  MoveC 1160 to (433.16, -30.09, -5) mm, rotated rx -180 ry 0 rz 30 deg; joints [33.705, -53.903, 150.227, 63.755, -91.912, 5.472] to (420.46, -17.39, -5) mm, rotated rx -180 ry 0 rz 30 deg; joints [33.923, -53.753, 148.985, 63.944, -91.411, 4.501]
  MoveL 1161 to (395.06, -17.39, -5) mm, rotated rx -180 ry 0 rz 0 deg; joints [25.034, -53.985, 155.724, 25.42, -99.757, 5.283]
  MoveL 1162 to (318.86, -17.39, -5) mm, rotated rx -180 ry 0 rz 0 deg; joints [22.969, -53.773, 150.895, 23.082, -95.687, 3.059]
  MoveC 1163 to (306.16, -30.09, -5) mm, rotated rx -180 ry 0 rz 0 deg; joints [21.911, -53.706, 150.409, 22.005, -95.348, 2.779] to (293.46, -17.39, -5) mm, rotated rx -180 ry 0 rz 0 deg; joints [22.351, -53.577, 149.245, 22.413, -94.372, 2.431]
  MoveL 1164 to (191.86, -17.39, -5) mm, rotated rx -180 ry 0 rz 0 deg; joints [20.165, -52.294, 142.446, 20.16, -89.274, 0.325]
  MoveC 1165 to (179.16, -30.09, -5) mm, rotated rx -180 ry 0 rz 0 deg; joints [19.25, -52.149, 141.884, 19.247, -88.88, 0.185] to (166.46, -17.39, -5) mm, rotated rx -180 ry 0 rz 0 deg; joints [19.681, -51.866, 140.698, 19.687, -88.03, -0.121]
  MoveL 1166 to (90.26, -17.39, -5) mm, rotated rx -180 ry 0 rz 0 deg; joints [18.355, -50.37, 135.332, 18.442, -84.349, -1.32]
  MoveL 1167 to (64.86, -17.39, -5) mm, rotated rx 180 ry 0 rz 0 deg; joints [17.951, -49.807, 133.502, 18.078, -83.134, -1.681]
  MoveC 1168 to (61.14, -26.37, -5) mm, rotated rx 180 ry 0 rz 0 deg; joints [17.461, -49.78, 133.439, 17.587, -83.082, -1.64] to (52.16, -30.09, -5) mm, rotated rx -180 ry 0 rz 0 deg; joints [17.147, -49.597, 132.868, 17.286, -82.702, -1.723]
  MoveL 1169 to (52.16, -30.09, -5) mm, rotated rx -180 ry 0 rz 0 deg; joints [17.147, -49.597, 132.868, 17.286, -82.702, -1.723]
  MoveC 1170 to (43.18, -26.37, -5) mm, rotated rx -180 ry 0 rz 0 deg; joints [17.193, -49.362, 132.128, 17.351, -82.221, -1.88] to (39.46, -17.39, -5) mm, rotated rx -180 ry 0 rz 0 deg; joints [17.563, -49.213, 131.65, 17.739, -81.923, -2.026]
  MoveL 1171 to (14.06, -17.39, -5) mm, rotated rx 180 ry 0 rz 0 deg; joints [17.191, -48.59, 129.776, 17.421, -80.714, -2.357]
  MoveC 1172 to (13.61, -17.2, -5) mm, rotated rx -180 ry 0 rz 0 deg; joints [17.194, -48.578, 129.738, 17.424, -80.69, -2.365] to (13.42, -16.75, -5) mm, rotated rx 180 ry 0 rz 0 deg; joints [17.212, -48.57, 129.714, 17.443, -80.675, -2.373]
  MoveL 1173 to (13.42, -16.12, -5) mm, rotated rx 180 ry 0 rz 0 deg; joints [17.241, -48.565, 129.7, 17.474, -80.667, -2.38]
  MoveC 1174 to (13.42, -15.67, -4.81) mm, rotated rx -180 ry 0 rz 0 deg; joints [17.262, -48.576, 129.692, 17.495, -80.65, -2.389] to (13.42, -15.48, -4.37) mm, rotated rx 180 ry 0 rz 0 deg; joints [17.27, -48.607, 129.693, 17.505, -80.622, -2.399]
  Set speed (1000.0 mm/s)
  MoveL 1175 to (13.42, -15.48, 5) mm, rotated rx -180 ry 0 rz 0 deg; joints [17.266, -49.29, 129.811, 17.53, -80.082, -2.572]
  MoveL 1176 to (12.15, -16.75, 5) mm, rotated rx -180 ry 0 rz 0 deg; joints [17.189, -49.267, 129.745, 17.454, -80.039, -2.572]
  Set speed (25.4 mm/s)
  MoveL 1177 to (12.15, -16.75, 1) mm, rotated rx -180 ry 0 rz 0 deg; joints [17.191, -48.975, 129.696, 17.443, -80.27, -2.499]
  MoveL 1178 to (12.15, -16.75, -7.72) mm, rotated rx -180 ry 0 rz 0 deg; joints [17.195, -48.34, 129.584, 17.421, -80.77, -2.34]
  MoveC 1179 to (12.34, -16.75, -8.16) mm, rotated rx -180 ry 0 rz 0 deg; joints [17.198, -48.312, 129.592, 17.422, -80.804, -2.33] to (12.79, -16.75, -8.35) mm, rotated rx -180 ry 0 rz 0 deg; joints [17.204, -48.309, 129.623, 17.427, -80.836, -2.32]
  Set speed (50.8 mm/s)
  MoveL 1180 to (13.42, -16.75, -8.35) mm, rotated rx 180 ry 0 rz 0 deg; joints [17.213, -48.325, 129.67, 17.435, -80.867, -2.312]
  MoveC 1181 to (13.87, -16.94, -8.35) mm, rotated rx 180 ry 0 rz 0 deg; joints [17.211, -48.337, 129.708, 17.432, -80.891, -2.304] to (14.06, -17.39, -8.35) mm, rotated rx -180 ry 0 rz 0 deg; joints [17.193, -48.345, 129.732, 17.412, -80.905, -2.297]
  MoveL 1182 to (14.06, -169.79, -8.35) mm, rotated rx 180 ry 0 rz 0 deg; joints [9.89, -49.145, 132.47, 9.97, -82.555, -0.881]
  MoveL 1183 to (471.26, -169.79, -8.35) mm, rotated rx 180 ry 0 rz 30 deg; joints [26.891, -53.506, 157.289, 57.471, -96.607, 11.391]
  MoveL 1184 to (471.26, -17.39, -8.35) mm, rotated rx 180 ry 0 rz 30 deg; joints [35.771, -53.739, 151.859, 65.871, -92.441, 7.208]
  MoveL 1185 to (445.86, -17.39, -8.35) mm, rotated rx 180 ry 0 rz 30 deg; joints [34.827, -53.598, 150.406, 64.887, -92.006, 5.964]
  MoveC 1186 to (433.16, -30.09, -8.35) mm, rotated rx -180 ry 0 rz 30 deg; joints [33.707, -53.551, 150.167, 63.767, -92.041, 5.734] to (420.46, -17.39, -8.35) mm, rotated rx -180 ry 0 rz 30 deg; joints [33.926, -53.411, 148.927, 63.953, -91.536, 4.756]
  MoveL 1187 to (395.06, -17.39, -8.35) mm, rotated rx -180 ry 0 rz 0 deg; joints [25.037, -53.585, 155.656, 25.448, -100.057, 5.428]
  MoveL 1188 to (318.86, -17.39, -8.35) mm, rotated rx -180 ry 0 rz 0 deg; joints [22.971, -53.416, 150.834, 23.097, -95.959, 3.176]
  MoveC 1189 to (306.16, -30.09, -8.35) mm, rotated rx 180 ry 0 rz 0 deg; joints [21.913, -53.353, 150.349, 22.018, -95.619, 2.89] to (293.46, -17.39, -8.35) mm, rotated rx -180 ry 0 rz 0 deg; joints [22.353, -53.232, 149.186, 22.423, -94.636, 2.54]
  MoveL 1190 to (191.86, -17.39, -8.35) mm, rotated rx 180 ry 0 rz 0 deg; joints [20.167, -51.993, 142.395, 20.161, -89.507, 0.411]
  MoveC 1191 to (179.16, -30.09, -8.35) mm, rotated rx -180 ry 0 rz 0 deg; joints [19.251, -51.851, 141.833, 19.247, -89.113, 0.266] to (166.46, -17.39, -8.35) mm, rotated rx -180 ry 0 rz 0 deg; joints [19.683, -51.575, 140.647, 19.686, -88.257, -0.04]
  MoveL 1192 to (90.26, -17.39, -8.35) mm, rotated rx -180 ry 0 rz 0 deg; joints [18.357, -50.104, 135.285, 18.436, -84.557, -1.25]
  MoveL 1193 to (64.86, -17.39, -8.35) mm, rotated rx -180 ry 0 rz 0 deg; joints [17.952, -49.548, 133.456, 18.072, -83.337, -1.614]
  MoveC 1194 to (61.14, -26.37, -8.35) mm, rotated rx -180 ry 0 rz 0 deg; joints [17.462, -49.522, 133.393, 17.581, -83.285, -1.576] to (52.16, -30.09, -8.35) mm, rotated rx -180 ry 0 rz 0 deg; joints [17.149, -49.341, 132.823, 17.279, -82.904, -1.66]
  MoveL 1195 to (52.16, -30.09, -8.35) mm, rotated rx -180 ry 0 rz 0 deg; joints [17.149, -49.341, 132.823, 17.279, -82.904, -1.66]
  MoveC 1196 to (43.18, -26.37, -8.35) mm, rotated rx -180 ry 0 rz 0 deg; joints [17.194, -49.108, 132.082, 17.344, -82.42, -1.818] to (39.46, -17.39, -8.35) mm, rotated rx -180 ry 0 rz 0 deg; joints [17.565, -48.961, 131.605, 17.731, -82.12, -1.963]
  MoveL 1197 to (14.06, -17.39, -8.35) mm, rotated rx 180 ry 0 rz 0 deg; joints [17.193, -48.345, 129.732, 17.412, -80.905, -2.297]
  MoveC 1198 to (13.61, -17.2, -8.35) mm, rotated rx -180 ry 0 rz 0 deg; joints [17.195, -48.333, 129.694, 17.416, -80.881, -2.305] to (13.42, -16.75, -8.35) mm, rotated rx 180 ry 0 rz 0 deg; joints [17.213, -48.325, 129.67, 17.435, -80.867, -2.312]
  MoveL 1199 to (13.42, -16.12, -8.35) mm, rotated rx -180 ry 0 rz 0 deg; joints [17.243, -48.32, 129.656, 17.465, -80.858, -2.32]
  MoveC 1200 to (13.42, -15.67, -8.16) mm, rotated rx -180 ry 0 rz 0 deg; joints [17.263, -48.331, 129.648, 17.487, -80.842, -2.328] to (13.42, -15.48, -7.72) mm, rotated rx -180 ry 0 rz 0 deg; joints [17.272, -48.362, 129.649, 17.497, -80.814, -2.338]
  Set speed (1000.0 mm/s)
  MoveL 1201 to (13.42, -15.48, 6) mm, rotated rx 180 ry 0 rz 0 deg; joints [17.266, -49.363, 129.823, 17.533, -80.024, -2.59]
  MoveL 1202 to (-18.41, -15.48, 6) mm, rotated rx -180 ry 0 rz 0 deg; joints [16.82, -48.516, 127.438, 17.166, -78.533, -2.979]
  Set speed (25.4 mm/s)
  MoveL 1203 to (-18.41, -15.48, -4.37) mm, rotated rx -180 ry 0 rz 0 deg; joints [16.824, -47.785, 127.311, 17.136, -79.111, -2.798]
  MoveC 1204 to (-18.41, -15.67, -4.81) mm, rotated rx -180 ry 0 rz 0 deg; joints [16.816, -47.754, 127.31, 17.126, -79.138, -2.788] to (-18.41, -16.12, -5) mm, rotated rx -180 ry 0 rz 0 deg; joints [16.795, -47.745, 127.318, 17.104, -79.154, -2.779]
  Set speed (50.8 mm/s)
  MoveL 1205 to (-18.41, -16.75, -5) mm, rotated rx -180 ry 0 rz 0 deg; joints [16.767, -47.749, 127.332, 17.074, -79.162, -2.771]
  MoveC 1206 to (-18.6, -17.2, -5) mm, rotated rx 180 ry 0 rz 0 deg; joints [16.744, -47.748, 127.328, 17.051, -79.158, -2.768] to (-19.04, -17.39, -5) mm, rotated rx -180 ry 0 rz 0 deg; joints [16.729, -47.737, 127.299, 17.037, -79.139, -2.771]
  MoveL 1207 to (-39.46, -17.39, -5) mm, rotated rx -180 ry 0 rz 0 deg; joints [16.456, -47.188, 125.751, 16.818, -78.168, -3.017]
  MoveC 1208 to (-52.16, -30.09, -5) mm, rotated rx 180 ry 0 rz 0 deg; joints [15.728, -46.931, 125.057, 16.101, -77.708, -2.999] to (-64.86, -17.39, -5) mm, rotated rx -180 ry 0 rz 0 deg; joints [16.128, -46.481, 123.801, 16.561, -76.959, -3.315]
  MoveL 1209 to (-90.26, -17.39, -5) mm, rotated rx -180 ry 0 rz 0 deg; joints [15.813, -45.748, 121.826, 16.323, -75.747, -3.606]
  MoveL 1210 to (-166.46, -17.39, -5) mm, rotated rx -180 ry 0 rz 0 deg; joints [14.935, -43.396, 115.729, 15.709, -72.082, -4.442]
  MoveC 1211 to (-179.16, -30.09, -5) mm, rotated rx 180 ry 0 rz 0 deg; joints [14.282, -43.083, 114.956, 15.064, -71.585, -4.366] to (-191.86, -17.39, -5) mm, rotated rx -180 ry 0 rz 0 deg; joints [14.663, -42.561, 113.635, 15.537, -70.846, -4.712]
  MoveL 1212 to (-293.46, -17.39, -5) mm, rotated rx -180 ry 0 rz 0 deg; joints [13.666, -38.954, 104.895, 15.006, -65.798, -5.788]
  MoveC 1213 to (-306.16, -30.09, -5) mm, rotated rx -180 ry 0 rz 0 deg; joints [13.075, -38.58, 104.026, 14.418, -65.257, -5.668] to (-318.86, -17.39, -5) mm, rotated rx -180 ry 0 rz 0 deg; joints [13.438, -37.982, 102.606, 14.913, -64.502, -6.06]
  MoveL 1214 to (-395.06, -17.39, -5) mm, rotated rx -180 ry 0 rz 0 deg; joints [12.794, -34.878, 95.441, 14.734, -60.499, -6.909]
  MoveL 1215 to (-420.46, -17.39, -5) mm, rotated rx -180 ry 0 rz 0 deg; joints [12.593, -33.776, 92.938, 14.71, -59.119, -7.208]
  MoveC 1216 to (-433.16, -30.09, -5) mm, rotated rx -180 ry 0 rz 0 deg; joints [12.054, -33.329, 91.94, 14.168, -58.516, -7.053] to (-445.86, -17.39, -5) mm, rotated rx 180 ry 0 rz 0 deg; joints [12.398, -32.635, 90.369, 14.706, -57.712, -7.518]
  MoveL 1217 to (-471.26, -17.39, -5) mm, rotated rx -180 ry 0 rz 0 deg; joints [12.209, -31.453, 87.727, 14.724, -56.273, -7.841]
  MoveL 1218 to (-471.26, -169.79, -5) mm, rotated rx 180 ry 0 rz 0 deg; joints [6.952, -32.605, 90.415, 8.272, -57.207, -4.124]
  MoveL 1219 to (-14.06, -169.79, -5) mm, rotated rx -180 ry 0 rz 0 deg; joints [9.653, -48.705, 130.382, 9.771, -80.926, -1.136]
  MoveL 1220 to (-14.06, -17.39, -5) mm, rotated rx 180 ry 0 rz 0 deg; joints [16.797, -47.869, 127.675, 17.093, -79.377, -2.71]
  MoveL 1221 to (-19.04, -17.39, -5) mm, rotated rx -180 ry 0 rz 0 deg; joints [16.729, -47.737, 127.299, 17.037, -79.139, -2.771]
  MoveC 1222 to (-19.49, -17.2, -5) mm, rotated rx -180 ry 0 rz 0 deg; joints [16.732, -47.724, 127.26, 17.041, -79.116, -2.779] to (-19.68, -16.75, -5) mm, rotated rx -180 ry 0 rz 0 deg; joints [16.749, -47.716, 127.236, 17.06, -79.101, -2.787]
  MoveL 1223 to (-19.68, -16.12, -5) mm, rotated rx -180 ry 0 rz 0 deg; joints [16.778, -47.711, 127.222, 17.09, -79.094, -2.795]
  MoveC 1224 to (-19.68, -15.67, -4.81) mm, rotated rx -180 ry 0 rz 0 deg; joints [16.798, -47.721, 127.214, 17.111, -79.078, -2.804] to (-19.68, -15.48, -4.37) mm, rotated rx -180 ry 0 rz 0 deg; joints [16.807, -47.751, 127.216, 17.121, -79.051, -2.814]
  Set speed (1000.0 mm/s)
  MoveL 1225 to (-19.68, -15.48, 5) mm, rotated rx -180 ry 0 rz 0 deg; joints [16.803, -48.411, 127.33, 17.149, -78.529, -2.977]
  MoveL 1226 to (-18.41, -15.48, 5) mm, rotated rx -180 ry 0 rz 0 deg; joints [16.82, -48.446, 127.426, 17.163, -78.589, -2.962]
  Set speed (25.4 mm/s)
  MoveL 1227 to (-18.41, -15.48, 1) mm, rotated rx -180 ry 0 rz 0 deg; joints [16.822, -48.164, 127.378, 17.151, -78.813, -2.892]
  MoveL 1228 to (-18.41, -15.48, -7.71) mm, rotated rx -180 ry 0 rz 0 deg; joints [16.825, -47.548, 127.268, 17.126, -79.296, -2.74]
  MoveC 1229 to (-18.41, -15.67, -8.16) mm, rotated rx -180 ry 0 rz 0 deg; joints [16.817, -47.518, 127.267, 17.116, -79.324, -2.73] to (-18.41, -16.12, -8.35) mm, rotated rx 180 ry 0 rz 0 deg; joints [16.797, -47.508, 127.275, 17.095, -79.339, -2.721]
  Set speed (50.8 mm/s)
  MoveL 1230 to (-18.41, -16.75, -8.35) mm, rotated rx -180 ry 0 rz 0 deg; joints [16.768, -47.512, 127.289, 17.065, -79.347, -2.714]
  MoveC 1231 to (-18.6, -17.2, -8.35) mm, rotated rx -180 ry 0 rz 0 deg; joints [16.745, -47.511, 127.285, 17.042, -79.344, -2.71] to (-19.04, -17.39, -8.35) mm, rotated rx -180 ry 0 rz 0 deg; joints [16.731, -47.5, 127.255, 17.028, -79.325, -2.713]
  MoveL 1232 to (-39.46, -17.39, -8.35) mm, rotated rx -180 ry 0 rz 0 deg; joints [16.458, -46.956, 125.708, 16.808, -78.35, -2.961]
  MoveC 1233 to (-52.16, -30.09, -8.35) mm, rotated rx 180 ry 0 rz 0 deg; joints [15.729, -46.701, 125.015, 16.091, -77.889, -2.946] to (-64.86, -17.39, -8.35) mm, rotated rx 180 ry 0 rz 0 deg; joints [16.13, -46.255, 123.76, 16.551, -77.136, -3.262]
  MoveL 1234 to (-90.26, -17.39, -8.35) mm, rotated rx -180 ry 0 rz 0 deg; joints [15.814, -45.527, 121.785, 16.311, -75.919, -3.554]
  MoveL 1235 to (-166.46, -17.39, -8.35) mm, rotated rx -180 ry 0 rz 0 deg; joints [14.936, -43.19, 115.689, 15.696, -72.242, -4.395]
  MoveC 1236 to (-179.16, -30.09, -8.35) mm, rotated rx -180 ry 0 rz 0 deg; joints [14.283, -42.879, 114.917, 15.051, -71.744, -4.321] to (-191.86, -17.39, -8.35) mm, rotated rx 180 ry 0 rz 0 deg; joints [14.664, -42.359, 113.595, 15.523, -71.003, -4.667]
  MoveL 1237 to (-293.46, -17.39, -8.35) mm, rotated rx 180 ry 0 rz 0 deg; joints [13.667, -38.767, 104.856, 14.99, -65.941, -5.746]
  MoveC 1238 to (-306.16, -30.09, -8.35) mm, rotated rx -180 ry 0 rz 0 deg; joints [13.076, -38.395, 103.987, 14.402, -65.399, -5.628] to (-318.86, -17.39, -8.35) mm, rotated rx 180 ry 0 rz 0 deg; joints [13.439, -37.799, 102.568, 14.897, -64.641, -6.02]
  MoveL 1239 to (-395.06, -17.39, -8.35) mm, rotated rx 180 ry 0 rz 0 deg; joints [12.795, -34.705, 95.402, 14.716, -60.629, -6.87]
  MoveL 1240 to (-420.46, -17.39, -8.35) mm, rotated rx -180 ry 0 rz 0 deg; joints [12.594, -33.605, 92.899, 14.691, -59.246, -7.169]
  MoveC 1241 to (-433.16, -30.09, -8.35) mm, rotated rx -180 ry 0 rz 0 deg; joints [12.055, -33.16, 91.901, 14.15, -58.642, -7.016] to (-445.86, -17.39, -8.35) mm, rotated rx 180 ry 0 rz 0 deg; joints [12.399, -32.467, 90.33, 14.687, -57.836, -7.48]
  MoveL 1242 to (-471.26, -17.39, -8.35) mm, rotated rx 180 ry 0 rz 0 deg; joints [12.21, -31.288, 87.687, 14.703, -56.395, -7.803]
  MoveL 1243 to (-471.26, -169.79, -8.35) mm, rotated rx 180 ry 0 rz 0 deg; joints [6.952, -32.437, 90.375, 8.261, -57.334, -4.103]
  MoveL 1244 to (-14.06, -169.79, -8.35) mm, rotated rx 180 ry 0 rz 0 deg; joints [9.654, -48.458, 130.338, 9.767, -81.126, -1.101]
  MoveL 1245 to (-14.06, -17.39, -8.35) mm, rotated rx -180 ry 0 rz 0 deg; joints [16.799, -47.631, 127.631, 17.084, -79.563, -2.652]
  MoveL 1246 to (-19.04, -17.39, -8.35) mm, rotated rx -180 ry 0 rz 0 deg; joints [16.731, -47.5, 127.255, 17.028, -79.325, -2.713]
  MoveC 1247 to (-19.49, -17.2, -8.35) mm, rotated rx 180 ry 0 rz 0 deg; joints [16.733, -47.487, 127.217, 17.032, -79.301, -2.721] to (-19.68, -16.75, -8.35) mm, rotated rx -180 ry 0 rz 0 deg; joints [16.751, -47.479, 127.193, 17.051, -79.287, -2.729]
  MoveL 1248 to (-19.68, -16.12, -8.35) mm, rotated rx -180 ry 0 rz 0 deg; joints [16.78, -47.474, 127.179, 17.08, -79.279, -2.737]
  MoveC 1249 to (-19.68, -15.67, -8.16) mm, rotated rx -180 ry 0 rz 0 deg; joints [16.8, -47.484, 127.171, 17.102, -79.263, -2.746] to (-19.68, -15.48, -7.72) mm, rotated rx -180 ry 0 rz 0 deg; joints [16.808, -47.515, 127.173, 17.112, -79.236, -2.756]
  Set speed (1000.0 mm/s)
  MoveL 1250 to (-19.68, -15.48, 6) mm, rotated rx -180 ry 0 rz 0 deg; joints [16.802, -48.482, 127.342, 17.152, -78.473, -2.994]
  MoveL 1251 to (-13.42, -196.51, 6) mm, rotated rx -180 ry 0 rz 0 deg; joints [8.362, -49.629, 130.891, 8.475, -80.487, -1.011]
  Set speed (25.4 mm/s)
  MoveL 1252 to (-13.42, -196.51, -4.37) mm, rotated rx -180 ry 0 rz 0 deg; joints [8.366, -48.861, 130.76, 8.463, -81.116, -0.916]
  MoveC 1253 to (-13.42, -196.7, -4.81) mm, rotated rx -180 ry 0 rz 0 deg; joints [8.357, -48.829, 130.756, 8.453, -81.145, -0.911] to (-13.42, -197.15, -5) mm, rotated rx -180 ry 0 rz 0 deg; joints [8.335, -48.816, 130.759, 8.431, -81.159, -0.905]
  Set speed (50.8 mm/s)
  MoveL 1254 to (-13.42, -197.78, -5) mm, rotated rx -180 ry 0 rz 0 deg; joints [8.305, -48.818, 130.766, 8.4, -81.163, -0.9]
  MoveC 1255 to (-13.61, -198.23, -5) mm, rotated rx -180 ry 0 rz 0 deg; joints [8.281, -48.815, 130.757, 8.377, -81.157, -0.898] to (-14.06, -198.42, -5) mm, rotated rx 180 ry 0 rz 0 deg; joints [8.269, -48.804, 130.724, 8.365, -81.135, -0.899]
  MoveL 1256 to (-39.46, -198.42, -5) mm, rotated rx 180 ry 0 rz 0 deg; joints [8.094, -48.149, 128.771, 8.219, -79.848, -1.062]
  MoveC 1257 to (-52.16, -211.12, -5) mm, rotated rx -180 ry 0 rz 0 deg; joints [7.411, -47.85, 127.919, 7.538, -79.283, -1.024] to (-64.86, -198.42, -5) mm, rotated rx -180 ry 0 rz 0 deg; joints [7.926, -47.464, 126.796, 8.082, -78.565, -1.219]
  MoveL 1258 to (-90.26, -198.42, -5) mm, rotated rx -180 ry 0 rz 0 deg; joints [7.765, -46.752, 124.797, 7.956, -77.287, -1.371]
  MoveL 1259 to (-166.46, -198.42, -5) mm, rotated rx -180 ry 0 rz 0 deg; joints [7.318, -44.454, 118.646, 7.631, -73.455, -1.801]
  MoveC 1260 to (-179.16, -211.12, -5) mm, rotated rx -180 ry 0 rz 0 deg; joints [6.706, -44.093, 117.725, 7.014, -72.878, -1.7] to (-191.86, -198.42, -5) mm, rotated rx -180 ry 0 rz 0 deg; joints [7.18, -43.636, 116.54, 7.539, -72.173, -1.938]
  MoveL 1261 to (-293.46, -198.42, -5) mm, rotated rx 180 ry 0 rz 0 deg; joints [6.677, -40.095, 107.784, 7.253, -66.98, -2.475]
  MoveC 1262 to (-306.16, -211.12, -5) mm, rotated rx 180 ry 0 rz 0 deg; joints [6.123, -39.67, 106.774, 6.681, -66.373, -2.322] to (-318.86, -198.42, -5) mm, rotated rx 180 ry 0 rz 0 deg; joints [6.562, -39.14, 105.5, 7.201, -65.656, -2.609]
  MoveL 1263 to (-395.06, -198.42, -5) mm, rotated rx -180 ry 0 rz 0 deg; joints [6.24, -36.096, 98.375, 7.093, -61.589, -3.021]
  MoveL 1264 to (-420.46, -198.42, -5) mm, rotated rx -180 ry 0 rz 0 deg; joints [6.14, -35.016, 95.895, 7.074, -60.194, -3.164]
  MoveC 1265 to (-433.16, -211.12, -5) mm, rotated rx -180 ry 0 rz 0 deg; joints [5.633, -34.516, 94.762, 6.534, -59.536, -2.965] to (-445.86, -198.42, -5) mm, rotated rx 180 ry 0 rz 0 deg; joints [6.042, -33.9, 93.355, 7.065, -58.775, -3.312]
  MoveL 1266 to (-471.26, -198.42, -5) mm, rotated rx -180 ry 0 rz 0 deg; joints [5.948, -32.745, 90.749, 7.065, -57.328, -3.465]
  MoveL 1267 to (-471.26, -350.82, -5) mm, rotated rx -180 ry 0 rz 0 deg; joints [0.558, -33.102, 91.639, 0.655, -57.669, -0.07]
  MoveL 1268 to (-14.06, -350.82, -5) mm, rotated rx 180 ry 0 rz 0 deg; joints [0.777, -49.039, 131.64, 0.781, -81.732, 0.172]
  MoveL 1269 to (-14.06, -198.42, -5) mm, rotated rx 180 ry 0 rz 0 deg; joints [8.269, -48.804, 130.724, 8.365, -81.135, -0.899]
  MoveC 1270 to (-13.87, -197.97, -5) mm, rotated rx 180 ry 0 rz 0 deg; joints [8.292, -48.808, 130.734, 8.388, -81.142, -0.902] to (-13.42, -197.78, -5) mm, rotated rx -180 ry 0 rz 0 deg; joints [8.305, -48.818, 130.766, 8.4, -81.163, -0.9]
  MoveL 1271 to (-12.79, -197.79, -5) mm, rotated rx 180 ry 0 rz 0 deg; joints [8.309, -48.834, 130.815, 8.404, -81.196, -0.896]
  MoveC 1272 to (-12.34, -197.78, -4.81) mm, rotated rx -180 ry 0 rz 0 deg; joints [8.312, -48.859, 130.851, 8.407, -81.207, -0.895] to (-12.15, -197.78, -4.37) mm, rotated rx 180 ry 0 rz 0 deg; joints [8.313, -48.897, 130.871, 8.408, -81.189, -0.898]
  Set speed (1000.0 mm/s)
  MoveL 1273 to (-12.15, -197.78, 5) mm, rotated rx -180 ry 0 rz 0 deg; joints [8.31, -49.592, 130.991, 8.418, -80.62, -0.982]
  MoveL 1274 to (-13.42, -196.52, 5) mm, rotated rx -180 ry 0 rz 0 deg; joints [8.363, -49.555, 130.879, 8.474, -80.548, -1.001]
  Set speed (25.4 mm/s)
  MoveL 1275 to (-13.42, -196.51, 1) mm, rotated rx -180 ry 0 rz 0 deg; joints [8.364, -49.259, 130.829, 8.469, -80.791, -0.965]
  MoveL 1276 to (-13.42, -196.51, -7.71) mm, rotated rx -180 ry 0 rz 0 deg; joints [8.367, -48.613, 130.716, 8.46, -81.318, -0.886]
  MoveC 1277 to (-13.42, -196.7, -8.16) mm, rotated rx 180 ry 0 rz 0 deg; joints [8.358, -48.58, 130.712, 8.45, -81.346, -0.88] to (-13.42, -197.15, -8.35) mm, rotated rx -180 ry 0 rz 0 deg; joints [8.337, -48.568, 130.714, 8.428, -81.361, -0.875]
  Set speed (50.8 mm/s)
  MoveL 1278 to (-13.42, -197.78, -8.35) mm, rotated rx -180 ry 0 rz 0 deg; joints [8.306, -48.57, 130.721, 8.396, -81.365, -0.87]
  MoveC 1279 to (-13.61, -198.23, -8.35) mm, rotated rx 180 ry 0 rz 0 deg; joints [8.283, -48.566, 130.712, 8.373, -81.359, -0.868] to (-14.06, -198.42, -8.35) mm, rotated rx -180 ry 0 rz 0 deg; joints [8.27, -48.556, 130.68, 8.361, -81.337, -0.87]
  MoveL 1280 to (-39.46, -198.42, -8.35) mm, rotated rx 180 ry 0 rz 0 deg; joints [8.095, -47.907, 128.727, 8.215, -80.043, -1.034]
  MoveC 1281 to (-52.16, -211.12, -8.35) mm, rotated rx 180 ry 0 rz 0 deg; joints [7.412, -47.611, 127.875, 7.535, -79.477, -0.998] to (-64.86, -198.42, -8.35) mm, rotated rx -180 ry 0 rz 0 deg; joints [7.927, -47.229, 126.753, 8.078, -78.756, -1.192]
  MoveL 1282 to (-90.26, -198.42, -8.35) mm, rotated rx -180 ry 0 rz 0 deg; joints [7.766, -46.523, 124.754, 7.951, -77.472, -1.345]
  MoveL 1283 to (-166.46, -198.42, -8.35) mm, rotated rx -180 ry 0 rz 0 deg; joints [7.319, -44.241, 118.606, 7.625, -73.626, -1.777]
  MoveC 1284 to (-179.16, -211.12, -8.35) mm, rotated rx 180 ry 0 rz 0 deg; joints [6.707, -43.882, 117.684, 7.008, -73.047, -1.678] to (-191.86, -198.42, -8.35) mm, rotated rx -180 ry 0 rz 0 deg; joints [7.181, -43.427, 116.5, 7.533, -72.34, -1.916]
  MoveL 1285 to (-293.46, -198.42, -8.35) mm, rotated rx -180 ry 0 rz 0 deg; joints [6.678, -39.904, 107.745, 7.246, -67.131, -2.455]
  MoveC 1286 to (-306.16, -211.12, -8.35) mm, rotated rx -180 ry 0 rz 0 deg; joints [6.124, -39.48, 106.735, 6.674, -66.523, -2.303] to (-318.86, -198.42, -8.35) mm, rotated rx 180 ry 0 rz 0 deg; joints [6.563, -38.953, 105.462, 7.193, -65.803, -2.589]
  MoveL 1287 to (-395.06, -198.42, -8.35) mm, rotated rx -180 ry 0 rz 0 deg; joints [6.241, -35.919, 98.336, 7.085, -61.726, -3.002]
  MoveL 1288 to (-420.46, -198.42, -8.35) mm, rotated rx -180 ry 0 rz 0 deg; joints [6.14, -34.842, 95.857, 7.066, -60.328, -3.145]
  MoveC 1289 to (-433.16, -211.12, -8.35) mm, rotated rx 180 ry 0 rz 0 deg; joints [5.634, -34.343, 94.724, 6.526, -59.669, -2.948] to (-445.86, -198.42, -8.35) mm, rotated rx -180 ry 0 rz 0 deg; joints [6.043, -33.729, 93.316, 7.056, -58.906, -3.293]
  MoveL 1290 to (-471.26, -198.42, -8.35) mm, rotated rx -180 ry 0 rz 0 deg; joints [5.949, -32.578, 90.71, 7.056, -57.456, -3.447]
  MoveL 1291 to (-471.26, -350.82, -8.35) mm, rotated rx -180 ry 0 rz 0 deg; joints [0.559, -32.933, 91.6, 0.655, -57.799, -0.068]
  MoveL 1292 to (-14.06, -350.82, -8.35) mm, rotated rx -180 ry 0 rz 0 deg; joints [0.778, -48.788, 131.595, 0.781, -81.938, 0.175]
  MoveL 1293 to (-14.06, -198.42, -8.35) mm, rotated rx -180 ry 0 rz 0 deg; joints [8.27, -48.556, 130.68, 8.361, -81.337, -0.87]
  MoveC 1294 to (-13.87, -197.97, -8.35) mm, rotated rx -180 ry 0 rz 0 deg; joints [8.293, -48.559, 130.689, 8.385, -81.343, -0.872] to (-13.42, -197.79, -8.35) mm, rotated rx -180 ry 0 rz 0 deg; joints [8.306, -48.57, 130.721, 8.396, -81.365, -0.87]
  MoveL 1295 to (-12.79, -197.79, -8.35) mm, rotated rx 180 ry 0 rz 0 deg; joints [8.31, -48.585, 130.77, 8.4, -81.397, -0.866]
  MoveC 1296 to (-12.34, -197.78, -8.16) mm, rotated rx -180 ry 0 rz 0 deg; joints [8.313, -48.611, 130.807, 8.403, -81.409, -0.865] to (-12.15, -197.79, -7.72) mm, rotated rx -180 ry 0 rz 0 deg; joints [8.314, -48.649, 130.827, 8.405, -81.392, -0.868]
  Set speed (1000.0 mm/s)
  MoveL 1297 to (-12.15, -197.79, 6) mm, rotated rx 180 ry 0 rz 0 deg; joints [8.31, -49.667, 131.003, 8.42, -80.559, -0.992]
  MoveL 1298 to (12.15, -197.78, 6) mm, rotated rx -180 ry 0 rz 0 deg; joints [8.486, -50.287, 132.853, 8.569, -81.779, -0.832]
  Set speed (25.4 mm/s)
  MoveL 1299 to (12.15, -197.79, -4.37) mm, rotated rx -180 ry 0 rz 0 deg; joints [8.489, -49.496, 132.719, 8.559, -82.428, -0.734]
  MoveC 1300 to (12.34, -197.78, -4.81) mm, rotated rx -180 ry 0 rz 0 deg; joints [8.491, -49.466, 132.727, 8.56, -82.465, -0.729] to (12.79, -197.79, -5) mm, rotated rx -180 ry 0 rz 0 deg; joints [8.494, -49.463, 132.758, 8.563, -82.5, -0.724]
  Set speed (50.8 mm/s)
  MoveL 1301 to (13.42, -197.78, -5) mm, rotated rx 180 ry 0 rz 0 deg; joints [8.499, -49.478, 132.806, 8.567, -82.532, -0.719]
  MoveC 1302 to (13.87, -197.97, -5) mm, rotated rx 180 ry 0 rz 0 deg; joints [8.493, -49.49, 132.842, 8.561, -82.557, -0.715] to (14.06, -198.42, -5) mm, rotated rx -180 ry 0 rz 0 deg; joints [8.472, -49.495, 132.862, 8.539, -82.569, -0.711]
  MoveL 1303 to (14.06, -350.82, -5) mm, rotated rx -180 ry 0 rz 0 deg; joints [0.796, -49.719, 133.789, 0.798, -83.201, 0.19]
  MoveL 1304 to (471.26, -350.82, -5) mm, rotated rx 180 ry 0 rz -60 deg; joints [-17.821, -53.492, 151.801, -77.92, -91.55, -7.234]
  MoveL 1305 to (471.26, -198.42, -5) mm, rotated rx -180 ry 0 rz -60 deg; joints [-7.953, -53.613, 154.17, -68.26, -93.747, -8.91]
  MoveL 1306 to (445.86, -198.42, -5) mm, rotated rx 180 ry 0 rz -60 deg; joints [-7.722, -53.554, 152.428, -67.938, -93.155, -7.331]
  MoveC 1307 to (433.16, -211.12, -5) mm, rotated rx -180 ry 0 rz -60 deg; joints [-8.425, -53.482, 151.427, -68.591, -92.716, -6.505] to (420.46, -198.42, -5) mm, rotated rx 180 ry 0 rz -60 deg; joints [-7.503, -53.419, 150.671, -67.646, -92.571, -5.816]
  MoveL 1308 to (395.06, -198.42, -5) mm, rotated rx -180 ry 0 rz -30 deg; joints [0.221, -53.49, 157.85, -30.495, -101.818, -6.56]
  MoveL 1309 to (318.86, -198.42, -5) mm, rotated rx -180 ry 0 rz 0 deg; joints [11.533, -53.788, 154.611, 11.698, -99.734, 2.455]
  MoveC 1310 to (306.16, -211.12, -5) mm, rotated rx -180 ry 0 rz 0 deg; joints [10.523, -53.768, 153.917, 10.654, -99.108, 2.14] to (293.46, -198.42, -5) mm, rotated rx 180 ry 0 rz 0 deg; joints [11.197, -53.742, 152.89, 11.306, -98.104, 2.059]
  MoveL 1311 to (191.86, -198.42, -5) mm, rotated rx -180 ry 0 rz 0 deg; joints [10.026, -52.868, 145.843, 10.027, -92.06, 0.79]
  MoveC 1312 to (179.16, -211.12, -5) mm, rotated rx -180 ry 0 rz 0 deg; joints [9.162, -52.716, 145.093, 9.16, -91.478, 0.651] to (166.46, -198.42, -5) mm, rotated rx -180 ry 0 rz 0 deg; joints [9.77, -52.509, 144.04, 9.766, -90.639, 0.532]
  MoveL 1313 to (90.26, -198.42, -5) mm, rotated rx -180 ry 0 rz 0 deg; joints [9.076, -51.17, 138.532, 9.087, -86.526, -0.144]
  MoveL 1314 to (64.86, -198.42, -5) mm, rotated rx -180 ry 0 rz 0 deg; joints [8.865, -50.646, 136.661, 8.892, -85.193, -0.343]
  MoveC 1315 to (61.14, -207.4, -5) mm, rotated rx 180 ry 0 rz 0 deg; joints [8.37, -50.59, 136.485, 8.396, -85.069, -0.327] to (52.16, -211.12, -5) mm, rotated rx -180 ry 0 rz 0 deg; joints [8.111, -50.405, 135.857, 8.141, -84.629, -0.371]
  MoveL 1316 to (52.16, -211.12, -5) mm, rotated rx -180 ry 0 rz 0 deg; joints [8.111, -50.405, 135.857, 8.141, -84.629, -0.371]
  MoveC 1317 to (43.18, -207.4, -5) mm, rotated rx 180 ry 0 rz 0 deg; joints [8.235, -50.196, 135.148, 8.274, -84.135, -0.453] to (39.46, -198.42, -5) mm, rotated rx -180 ry 0 rz 0 deg; joints [8.664, -50.087, 134.771, 8.709, -83.875, -0.532]
  MoveL 1318 to (14.06, -198.42, -5) mm, rotated rx -180 ry 0 rz 0 deg; joints [8.472, -49.495, 132.862, 8.539, -82.569, -0.711]
  MoveC 1319 to (13.61, -198.23, -5) mm, rotated rx -180 ry 0 rz 0 deg; joints [8.478, -49.484, 132.825, 8.546, -82.545, -0.715] to (13.42, -197.79, -5) mm, rotated rx 180 ry 0 rz 0 deg; joints [8.499, -49.478, 132.806, 8.567, -82.532, -0.719]
  MoveL 1320 to (13.42, -197.15, -5) mm, rotated rx -180 ry 0 rz 0 deg; joints [8.531, -49.476, 132.799, 8.599, -82.528, -0.724]
  MoveC 1321 to (13.42, -196.7, -4.81) mm, rotated rx 180 ry 0 rz 0 deg; joints [8.553, -49.489, 132.797, 8.622, -82.513, -0.729] to (13.42, -196.52, -4.37) mm, rotated rx -180 ry 0 rz 0 deg; joints [8.562, -49.523, 132.801, 8.631, -82.484, -0.734]
  Set speed (1000.0 mm/s)
  MoveL 1322 to (13.42, -196.51, 5) mm, rotated rx 180 ry 0 rz 0 deg; joints [8.559, -50.238, 132.922, 8.64, -81.897, -0.824]
  MoveL 1323 to (12.15, -197.79, 5) mm, rotated rx 180 ry 0 rz 0 deg; joints [8.486, -50.21, 132.84, 8.568, -81.842, -0.823]
  Set speed (25.4 mm/s)
  MoveL 1324 to (12.15, -197.79, 1) mm, rotated rx 180 ry 0 rz 0 deg; joints [8.488, -49.906, 132.79, 8.564, -82.093, -0.785]
  MoveL 1325 to (12.15, -197.78, -7.72) mm, rotated rx -180 ry 0 rz 0 deg; joints [8.491, -49.24, 132.673, 8.557, -82.636, -0.703]
  MoveC 1326 to (12.34, -197.79, -8.16) mm, rotated rx 180 ry 0 rz 0 deg; joints [8.492, -49.211, 132.681, 8.557, -82.673, -0.697] to (12.79, -197.79, -8.35) mm, rotated rx -180 ry 0 rz 0 deg; joints [8.495, -49.207, 132.713, 8.56, -82.708, -0.692]
  Set speed (50.8 mm/s)
  MoveL 1327 to (13.42, -197.78, -8.35) mm, rotated rx -180 ry 0 rz 0 deg; joints [8.5, -49.222, 132.761, 8.564, -82.74, -0.688]
  MoveC 1328 to (13.87, -197.97, -8.35) mm, rotated rx 180 ry 0 rz 0 deg; joints [8.494, -49.233, 132.797, 8.558, -82.765, -0.684] to (14.06, -198.42, -8.35) mm, rotated rx -180 ry 0 rz 0 deg; joints [8.473, -49.239, 132.816, 8.536, -82.778, -0.679]
  MoveL 1329 to (14.06, -350.82, -8.35) mm, rotated rx -180 ry 0 rz 0 deg; joints [0.797, -49.459, 133.742, 0.798, -83.415, 0.193]
  MoveL 1330 to (471.26, -350.82, -8.35) mm, rotated rx 180 ry 0 rz -60 deg; joints [-17.821, -53.128, 151.739, -77.929, -91.613, -7.53]
  MoveL 1331 to (471.26, -198.42, -8.35) mm, rotated rx -180 ry 0 rz -60 deg; joints [-7.952, -53.228, 154.104, -68.28, -93.865, -9.207]
  MoveL 1332 to (445.86, -198.42, -8.35) mm, rotated rx -180 ry 0 rz -60 deg; joints [-7.721, -53.184, 152.365, -67.953, -93.271, -7.615]
  MoveC 1333 to (433.16, -211.12, -8.35) mm, rotated rx -180 ry 0 rz -60 deg; joints [-8.424, -53.121, 151.366, -68.604, -92.825, -6.784] to (420.46, -198.42, -8.35) mm, rotated rx -180 ry 0 rz -60 deg; joints [-7.503, -53.064, 150.61, -67.658, -92.683, -6.088]
  MoveL 1334 to (395.06, -198.42, -8.35) mm, rotated rx -180 ry 0 rz -30 deg; joints [0.223, -53.068, 157.777, -30.531, -102.12, -6.741]
  MoveL 1335 to (318.86, -198.42, -8.35) mm, rotated rx -180 ry 0 rz 0 deg; joints [11.534, -53.398, 154.545, 11.711, -100.05, 2.521]
  MoveC 1336 to (306.16, -211.12, -8.35) mm, rotated rx 180 ry 0 rz 0 deg; joints [10.525, -53.385, 153.852, 10.665, -99.42, 2.199] to (293.46, -198.42, -8.35) mm, rotated rx -180 ry 0 rz 0 deg; joints [11.198, -53.368, 152.826, 11.316, -98.408, 2.12]
  MoveL 1337 to (191.86, -198.42, -8.35) mm, rotated rx -180 ry 0 rz 0 deg; joints [10.028, -52.547, 145.788, 10.031, -92.322, 0.837]
  MoveC 1338 to (179.16, -211.12, -8.35) mm, rotated rx -180 ry 0 rz 0 deg; joints [9.163, -52.4, 145.039, 9.163, -91.736, 0.693] to (166.46, -198.42, -8.35) mm, rotated rx -180 ry 0 rz 0 deg; joints [9.772, -52.2, 143.987, 9.768, -90.892, 0.576]
  MoveL 1339 to (90.26, -198.42, -8.35) mm, rotated rx -180 ry 0 rz 0 deg; joints [9.077, -50.889, 138.483, 9.086, -86.755, -0.108]
  MoveL 1340 to (64.86, -198.42, -8.35) mm, rotated rx 180 ry 0 rz 0 deg; joints [8.866, -50.374, 136.613, 8.89, -85.415, -0.308]
  MoveC 1341 to (61.14, -207.4, -8.35) mm, rotated rx -180 ry 0 rz 0 deg; joints [8.371, -50.319, 136.437, 8.395, -85.291, -0.294] to (52.16, -211.12, -8.35) mm, rotated rx -180 ry 0 rz 0 deg; joints [8.112, -50.136, 135.81, 8.14, -84.848, -0.34]
  MoveL 1342 to (52.16, -211.12, -8.35) mm, rotated rx -180 ry 0 rz 0 deg; joints [8.112, -50.136, 135.81, 8.14, -84.848, -0.34]
  MoveC 1343 to (43.18, -207.4, -8.35) mm, rotated rx -180 ry 0 rz 0 deg; joints [8.236, -49.93, 135.101, 8.272, -84.351, -0.422] to (39.46, -198.42, -8.35) mm, rotated rx 180 ry 0 rz 0 deg; joints [8.665, -49.823, 134.724, 8.707, -84.09, -0.499]
  MoveL 1344 to (14.06, -198.42, -8.35) mm, rotated rx 180 ry 0 rz 0 deg; joints [8.473, -49.239, 132.816, 8.536, -82.778, -0.679]
  MoveC 1345 to (13.61, -198.23, -8.35) mm, rotated rx 180 ry 0 rz 0 deg; joints [8.479, -49.228, 132.78, 8.543, -82.753, -0.684] to (13.42, -197.78, -8.35) mm, rotated rx -180 ry 0 rz 0 deg; joints [8.5, -49.222, 132.761, 8.564, -82.74, -0.688]
  MoveL 1346 to (13.42, -197.15, -8.35) mm, rotated rx -180 ry 0 rz 0 deg; joints [8.532, -49.22, 132.754, 8.596, -82.736, -0.692]
  MoveC 1347 to (13.42, -196.7, -8.16) mm, rotated rx -180 ry 0 rz 0 deg; joints [8.554, -49.233, 132.751, 8.619, -82.721, -0.697] to (13.42, -196.52, -7.72) mm, rotated rx -180 ry 0 rz 0 deg; joints [8.563, -49.267, 132.755, 8.629, -82.692, -0.703]
  Set speed (1000.0 mm/s)
  MoveL 1348 to (13.42, -196.51, 6) mm, rotated rx -180 ry 0 rz 0 deg; joints [8.558, -50.314, 132.935, 8.641, -81.834, -0.834]
  MoveL 1349 to (12.15, -384.12, 6) mm, rotated rx 180 ry 0 rz 0 deg; joints [-0.896, -50.512, 133.784, -0.908, -82.403, 0.379]
  Set speed (25.4 mm/s)
  MoveL 1350 to (12.15, -384.12, -4.37) mm, rotated rx -180 ry 0 rz 0 deg; joints [-0.893, -49.71, 133.648, -0.904, -83.069, 0.368]
  MoveC 1351 to (12.34, -384.12, -4.81) mm, rotated rx 180 ry 0 rz 0 deg; joints [-0.893, -49.68, 133.656, -0.904, -83.107, 0.367] to (12.79, -384.12, -5) mm, rotated rx 180 ry 0 rz 0 deg; joints [-0.894, -49.676, 133.688, -0.904, -83.143, 0.367]
  Set speed (50.8 mm/s)
  MoveL 1352 to (13.42, -384.12, -5) mm, rotated rx 180 ry 0 rz 0 deg; joints [-0.894, -49.691, 133.736, -0.905, -83.176, 0.366]
  MoveC 1353 to (13.87, -384.31, -5) mm, rotated rx -180 ry 0 rz 0 deg; joints [-0.904, -49.701, 133.77, -0.914, -83.2, 0.367] to (14.06, -384.76, -5) mm, rotated rx -180 ry 0 rz 0 deg; joints [-0.927, -49.705, 133.783, -0.938, -83.209, 0.369]
  MoveL 1354 to (14.06, -537.16, -5) mm, rotated rx -180 ry 0 rz 0 deg; joints [-8.6, -49.363, 132.809, -8.675, -82.651, 1.259]
  MoveL 1355 to (471.26, -537.16, -5) mm, rotated rx -180 ry 0 rz -30 deg; joints [-25.099, -53.419, 157.939, -55.843, -97.643, -11.304]
  MoveL 1356 to (471.26, -384.76, -5) mm, rotated rx -180 ry 0 rz -60 deg; joints [-19.898, -53.432, 151.035, -79.962, -91.132, -6.597]
  MoveL 1357 to (445.86, -384.76, -5) mm, rotated rx -180 ry 0 rz -60 deg; joints [-19.356, -53.252, 149.354, -79.398, -90.927, -5.108]
  MoveC 1358 to (433.16, -397.46, -5) mm, rotated rx 180 ry 0 rz -60 deg; joints [-19.834, -53.098, 148.207, -79.86, -90.702, -4.139] to (420.46, -384.76, -5) mm, rotated rx -180 ry 0 rz -60 deg; joints [-18.843, -53.015, 147.654, -78.867, -90.698, -3.663]
  MoveL 1359 to (395.06, -384.76, -5) mm, rotated rx 180 ry 0 rz -30 deg; joints [-13.016, -53.543, 156.418, -43.654, -98.766, -8.178]
  MoveL 1360 to (318.86, -384.76, -5) mm, rotated rx 180 ry 0 rz 0 deg; joints [-1.271, -53.634, 155.738, -1.3, -101.232, 0]
  MoveC 1361 to (306.16, -397.46, -5) mm, rotated rx -180 ry 0 rz 0 deg; joints [-2.121, -53.647, 154.841, -2.16, -100.316, -0.147] to (293.46, -384.76, -5) mm, rotated rx -180 ry 0 rz 0 deg; joints [-1.233, -53.651, 153.994, -1.254, -99.471, 0.047]
  MoveL 1362 to (191.86, -384.76, -5) mm, rotated rx -180 ry 0 rz 0 deg; joints [-1.101, -52.945, 146.866, -1.107, -93.05, 0.197]
  MoveC 1363 to (179.16, -397.46, -5) mm, rotated rx -180 ry 0 rz 0 deg; joints [-1.841, -52.777, 145.933, -1.847, -92.286, 0.171] to (166.46, -384.76, -5) mm, rotated rx -180 ry 0 rz 0 deg; joints [-1.072, -52.614, 145.046, -1.077, -91.562, 0.227]
  MoveL 1364 to (90.26, -384.76, -5) mm, rotated rx -180 ry 0 rz 0 deg; joints [-0.994, -51.338, 139.492, -1, -87.285, 0.305]
  MoveL 1365 to (64.86, -384.76, -5) mm, rotated rx -180 ry 0 rz 0 deg; joints [-0.971, -50.829, 137.607, -0.977, -85.908, 0.327]
  MoveC 1366 to (61.14, -393.74, -5) mm, rotated rx -180 ry 0 rz 0 deg; joints [-1.443, -50.745, 137.315, -1.451, -85.702, 0.359] to (52.16, -397.46, -5) mm, rotated rx -180 ry 0 rz 0 deg; joints [-1.627, -50.551, 136.636, -1.636, -85.217, 0.384]
  MoveL 1367 to (52.16, -397.46, -5) mm, rotated rx -180 ry 0 rz 0 deg; joints [-1.627, -50.551, 136.636, -1.636, -85.217, 0.384]
  MoveC 1368 to (43.18, -393.74, -5) mm, rotated rx -180 ry 0 rz 0 deg; joints [-1.419, -50.359, 135.97, -1.429, -84.742, 0.382] to (39.46, -384.76, -5) mm, rotated rx 180 ry 0 rz 0 deg; joints [-0.948, -50.285, 135.704, -0.957, -84.551, 0.349]
  MoveL 1369 to (14.06, -384.76, -5) mm, rotated rx -180 ry 0 rz 0 deg; joints [-0.927, -49.705, 133.783, -0.938, -83.209, 0.369]
  MoveC 1370 to (13.61, -384.57, -5) mm, rotated rx 180 ry 0 rz 0 deg; joints [-0.917, -49.695, 133.749, -0.928, -83.186, 0.368] to (13.42, -384.12, -5) mm, rotated rx 180 ry 0 rz 0 deg; joints [-0.894, -49.691, 133.736, -0.905, -83.176, 0.366]
  MoveL 1371 to (13.42, -383.49, -5) mm, rotated rx -180 ry 0 rz 0 deg; joints [-0.862, -49.691, 133.737, -0.872, -83.176, 0.363]
  MoveC 1372 to (13.42, -383.04, -4.81) mm, rotated rx 180 ry 0 rz 0 deg; joints [-0.839, -49.706, 133.74, -0.849, -83.165, 0.361] to (13.42, -382.85, -4.37) mm, rotated rx -180 ry 0 rz 0 deg; joints [-0.83, -49.741, 133.746, -0.84, -83.136, 0.36]
  Set speed (1000.0 mm/s)
  MoveL 1373 to (13.42, -382.85, 5) mm, rotated rx -180 ry 0 rz 0 deg; joints [-0.832, -50.467, 133.869, -0.843, -82.534, 0.369]
  MoveL 1374 to (12.15, -384.12, 5) mm, rotated rx -180 ry 0 rz 0 deg; joints [-0.895, -50.435, 133.771, -0.907, -82.468, 0.378]
  Set speed (25.4 mm/s)
  MoveL 1375 to (12.15, -384.12, 1) mm, rotated rx -180 ry 0 rz 0 deg; joints [-0.895, -50.125, 133.719, -0.906, -82.725, 0.373]
  MoveL 1376 to (12.15, -384.12, -7.71) mm, rotated rx 180 ry 0 rz 0 deg; joints [-0.893, -49.451, 133.602, -0.903, -83.282, 0.364]
  MoveC 1377 to (12.34, -384.12, -8.16) mm, rotated rx -180 ry 0 rz 0 deg; joints [-0.893, -49.42, 133.61, -0.903, -83.321, 0.364] to (12.79, -384.12, -8.35) mm, rotated rx 180 ry 0 rz 0 deg; joints [-0.893, -49.416, 133.641, -0.903, -83.356, 0.363]
  Set speed (50.8 mm/s)
  MoveL 1378 to (13.42, -384.12, -8.35) mm, rotated rx -180 ry 0 rz 0 deg; joints [-0.893, -49.431, 133.69, -0.903, -83.39, 0.363]
  MoveC 1379 to (13.87, -384.31, -8.35) mm, rotated rx 180 ry 0 rz 0 deg; joints [-0.903, -49.441, 133.723, -0.913, -83.413, 0.363] to (14.06, -384.76, -8.35) mm, rotated rx -180 ry 0 rz 0 deg; joints [-0.926, -49.445, 133.737, -0.936, -83.423, 0.365]
  MoveL 1380 to (14.06, -537.16, -8.35) mm, rotated rx -180 ry 0 rz 0 deg; joints [-8.6, -49.107, 132.763, -8.671, -82.859, 1.227]
  MoveL 1381 to (471.26, -537.16, -8.35) mm, rotated rx -180 ry 0 rz -30 deg; joints [-25.099, -52.995, 157.866, -55.883, -97.84, -11.597]
  MoveL 1382 to (471.26, -384.76, -8.35) mm, rotated rx -180 ry 0 rz -60 deg; joints [-19.898, -53.074, 150.973, -79.968, -91.184, -6.889]
  MoveL 1383 to (445.86, -384.76, -8.35) mm, rotated rx -180 ry 0 rz -60 deg; joints [-19.357, -52.907, 149.295, -79.403, -90.979, -5.389]
  MoveC 1384 to (433.16, -397.46, -8.35) mm, rotated rx -180 ry 0 rz -60 deg; joints [-19.835, -52.761, 148.149, -79.864, -90.751, -4.414] to (420.46, -384.76, -8.35) mm, rotated rx -180 ry 0 rz -60 deg; joints [-18.843, -52.682, 147.597, -78.87, -90.751, -3.933]
  MoveL 1385 to (395.06, -384.76, -8.35) mm, rotated rx -180 ry 0 rz -30 deg; joints [-13.016, -53.136, 156.348, -43.69, -99.01, -8.414]
  MoveL 1386 to (318.86, -384.76, -8.35) mm, rotated rx -180 ry 0 rz 0 deg; joints [-1.27, -53.233, 155.67, -1.301, -101.564, -0.008]
  MoveC 1387 to (306.16, -397.46, -8.35) mm, rotated rx -180 ry 0 rz 0 deg; joints [-2.12, -53.256, 154.774, -2.161, -100.641, -0.159] to (293.46, -384.76, -8.35) mm, rotated rx -180 ry 0 rz 0 deg; joints [-1.232, -53.267, 153.928, -1.255, -99.789, 0.04]
  MoveL 1388 to (191.86, -384.76, -8.35) mm, rotated rx 180 ry 0 rz 0 deg; joints [-1.1, -52.617, 146.809, -1.106, -93.322, 0.191]
  MoveC 1389 to (179.16, -397.46, -8.35) mm, rotated rx -180 ry 0 rz 0 deg; joints [-1.84, -52.455, 145.878, -1.846, -92.552, 0.162] to (166.46, -384.76, -8.35) mm, rotated rx -180 ry 0 rz 0 deg; joints [-1.071, -52.298, 144.991, -1.076, -91.823, 0.222]
  MoveL 1390 to (90.26, -384.76, -8.35) mm, rotated rx 180 ry 0 rz 0 deg; joints [-0.994, -51.052, 139.442, -0.999, -87.52, 0.3]
  MoveL 1391 to (64.86, -384.76, -8.35) mm, rotated rx 180 ry 0 rz 0 deg; joints [-0.97, -50.553, 137.558, -0.976, -86.136, 0.323]
  MoveC 1392 to (61.14, -393.74, -8.35) mm, rotated rx -180 ry 0 rz 0 deg; joints [-1.442, -50.47, 137.266, -1.45, -85.928, 0.353] to (52.16, -397.46, -8.35) mm, rotated rx -180 ry 0 rz 0 deg; joints [-1.626, -50.279, 136.588, -1.635, -85.441, 0.378]
  MoveL 1393 to (52.16, -397.46, -8.35) mm, rotated rx -180 ry 0 rz 0 deg; joints [-1.626, -50.279, 136.588, -1.635, -85.441, 0.378]
  MoveC 1394 to (43.18, -393.74, -8.35) mm, rotated rx -180 ry 0 rz 0 deg; joints [-1.419, -50.09, 135.922, -1.428, -84.964, 0.376] to (39.46, -384.76, -8.35) mm, rotated rx -180 ry 0 rz 0 deg; joints [-0.948, -50.017, 135.657, -0.956, -84.771, 0.345]
  MoveL 1395 to (14.06, -384.76, -8.35) mm, rotated rx -180 ry 0 rz 0 deg; joints [-0.926, -49.445, 133.737, -0.936, -83.423, 0.365]
  MoveC 1396 to (13.61, -384.57, -8.35) mm, rotated rx 180 ry 0 rz 0 deg; joints [-0.916, -49.435, 133.703, -0.927, -83.399, 0.365] to (13.42, -384.12, -8.35) mm, rotated rx -180 ry 0 rz 0 deg; joints [-0.893, -49.431, 133.69, -0.903, -83.39, 0.363]
  MoveL 1397 to (13.42, -383.49, -8.35) mm, rotated rx 180 ry 0 rz 0 deg; joints [-0.861, -49.431, 133.69, -0.871, -83.39, 0.359]
  MoveC 1398 to (13.42, -383.04, -8.16) mm, rotated rx 180 ry 0 rz 0 deg; joints [-0.838, -49.446, 133.693, -0.848, -83.378, 0.357] to (13.42, -382.85, -7.72) mm, rotated rx -180 ry 0 rz 0 deg; joints [-0.829, -49.481, 133.7, -0.839, -83.35, 0.357]
  Set speed (1000.0 mm/s)
  MoveL 1399 to (13.42, -382.85, 6) mm, rotated rx -180 ry 0 rz 0 deg; joints [-0.832, -50.544, 133.882, -0.844, -82.469, 0.37]
  MoveL 1400 to (-13.42, -382.85, 6) mm, rotated rx 180 ry 0 rz 0 deg; joints [-0.813, -49.87, 131.827, -0.827, -81.089, 0.388]
  Set speed (25.4 mm/s)
  MoveL 1401 to (-13.42, -382.85, -4.37) mm, rotated rx -180 ry 0 rz 0 deg; joints [-0.811, -49.091, 131.694, -0.823, -81.734, 0.378]
  MoveC 1402 to (-13.42, -383.04, -4.81) mm, rotated rx 180 ry 0 rz 0 deg; joints [-0.82, -49.057, 131.688, -0.832, -81.762, 0.379] to (-13.42, -383.49, -5) mm, rotated rx -180 ry 0 rz 0 deg; joints [-0.842, -49.043, 131.685, -0.855, -81.773, 0.382]
  Set speed (50.8 mm/s)
  MoveL 1403 to (-13.42, -384.12, -5) mm, rotated rx -180 ry 0 rz 0 deg; joints [-0.873, -49.043, 131.684, -0.887, -81.773, 0.386]
  MoveC 1404 to (-13.61, -384.57, -5) mm, rotated rx -180 ry 0 rz 0 deg; joints [-0.895, -49.038, 131.669, -0.909, -81.763, 0.389] to (-14.06, -384.76, -5) mm, rotated rx -180 ry 0 rz 0 deg; joints [-0.904, -49.026, 131.635, -0.918, -81.74, 0.39]
  MoveL 1405 to (-39.46, -384.76, -5) mm, rotated rx 180 ry 0 rz 0 deg; joints [-0.885, -48.38, 129.672, -0.901, -80.423, 0.409]
  MoveC 1406 to (-52.16, -397.46, -5) mm, rotated rx -180 ry 0 rz 0 deg; joints [-1.484, -48.035, 128.661, -1.512, -79.76, 0.519] to (-64.86, -384.76, -5) mm, rotated rx -180 ry 0 rz 0 deg; joints [-0.866, -47.705, 127.687, -0.886, -79.114, 0.426]
  MoveL 1407 to (-90.26, -384.76, -5) mm, rotated rx -180 ry 0 rz 0 deg; joints [-0.848, -47.001, 125.681, -0.872, -77.812, 0.443]
  MoveL 1408 to (-166.46, -384.76, -5) mm, rotated rx 180 ry 0 rz 0 deg; joints [-0.799, -44.724, 119.512, -0.835, -73.92, 0.492]
  MoveC 1409 to (-179.16, -397.46, -5) mm, rotated rx 180 ry 0 rz 0 deg; joints [-1.341, -44.31, 118.44, -1.405, -73.265, 0.656] to (-191.86, -384.76, -5) mm, rotated rx -180 ry 0 rz 0 deg; joints [-0.783, -43.911, 117.401, -0.825, -72.622, 0.507]
  MoveL 1410 to (-293.46, -384.76, -5) mm, rotated rx 180 ry 0 rz 0 deg; joints [-0.728, -40.394, 108.637, -0.793, -67.376, 0.566]
  MoveC 1411 to (-306.16, -397.46, -5) mm, rotated rx -180 ry 0 rz 0 deg; joints [-1.223, -39.912, 107.481, -1.336, -66.705, 0.782] to (-318.86, -384.76, -5) mm, rotated rx -180 ry 0 rz 0 deg; joints [-0.715, -39.445, 106.354, -0.787, -66.041, 0.581]
  MoveL 1412 to (-395.06, -384.76, -5) mm, rotated rx -180 ry 0 rz 0 deg; joints [-0.679, -36.42, 99.238, -0.774, -61.95, 0.626]
  MoveL 1413 to (-420.46, -384.76, -5) mm, rotated rx 180 ry 0 rz 0 deg; joints [-0.668, -35.347, 96.764, -0.772, -60.549, 0.642]
  MoveC 1414 to (-433.16, -397.46, -5) mm, rotated rx -180 ry 0 rz 0 deg; joints [-1.124, -34.786, 95.484, -1.305, -59.835, 0.911] to (-445.86, -384.76, -5) mm, rotated rx -180 ry 0 rz 0 deg; joints [-0.657, -34.239, 94.231, -0.771, -59.125, 0.658]
  MoveL 1415 to (-471.26, -384.76, -5) mm, rotated rx -180 ry 0 rz 0 deg; joints [-0.647, -33.092, 91.634, -0.77, -57.674, 0.674]
  MoveL 1416 to (-471.26, -537.16, -5) mm, rotated rx 180 ry 0 rz 0 deg; joints [-6.036, -32.652, 90.701, -7.176, -57.379, 4.063]
  MoveL 1417 to (-14.06, -537.16, -5) mm, rotated rx -180 ry 0 rz 0 deg; joints [-8.394, -48.675, 130.673, -8.498, -81.214, 1.451]
  MoveL 1418 to (-14.06, -384.76, -5) mm, rotated rx -180 ry 0 rz 0 deg; joints [-0.904, -49.026, 131.635, -0.918, -81.74, 0.39]
  MoveC 1419 to (-13.87, -384.31, -5) mm, rotated rx -180 ry 0 rz 0 deg; joints [-0.882, -49.031, 131.649, -0.896, -81.75, 0.387] to (-13.42, -384.12, -5) mm, rotated rx -180 ry 0 rz 0 deg; joints [-0.873, -49.043, 131.684, -0.887, -81.773, 0.386]
  MoveL 1420 to (-12.79, -384.12, -5) mm, rotated rx -180 ry 0 rz 0 deg; joints [-0.874, -49.058, 131.733, -0.887, -81.806, 0.385]
  MoveC 1421 to (-12.34, -384.12, -4.81) mm, rotated rx -180 ry 0 rz 0 deg; joints [-0.874, -49.083, 131.77, -0.887, -81.818, 0.385] to (-12.15, -384.12, -4.37) mm, rotated rx 180 ry 0 rz 0 deg; joints [-0.874, -49.122, 131.79, -0.888, -81.8, 0.386]
  Set speed (1000.0 mm/s)
  MoveL 1422 to (-12.15, -384.12, 5) mm, rotated rx 180 ry 0 rz 0 deg; joints [-0.877, -49.826, 131.911, -0.891, -81.216, 0.395]
  MoveL 1423 to (-13.42, -382.85, 5) mm, rotated rx 180 ry 0 rz 0 deg; joints [-0.813, -49.795, 131.815, -0.827, -81.151, 0.387]
  Set speed (25.4 mm/s)
  MoveL 1424 to (-13.42, -382.85, 1) mm, rotated rx 180 ry 0 rz 0 deg; joints [-0.812, -49.494, 131.764, -0.825, -81.401, 0.383]
  MoveL 1425 to (-13.42, -382.85, -7.71) mm, rotated rx -180 ry 0 rz 0 deg; joints [-0.81, -48.839, 131.649, -0.822, -81.941, 0.375]
  MoveC 1426 to (-13.42, -383.04, -8.16) mm, rotated rx -180 ry 0 rz 0 deg; joints [-0.819, -48.805, 131.643, -0.831, -81.969, 0.376] to (-13.42, -383.49, -8.35) mm, rotated rx -180 ry 0 rz 0 deg; joints [-0.841, -48.791, 131.64, -0.854, -81.98, 0.379]
  Set speed (50.8 mm/s)
  MoveL 1427 to (-13.42, -384.12, -8.35) mm, rotated rx -180 ry 0 rz 0 deg; joints [-0.873, -48.791, 131.639, -0.885, -81.98, 0.383]
  MoveC 1428 to (-13.61, -384.57, -8.35) mm, rotated rx 180 ry 0 rz 0 deg; joints [-0.895, -48.786, 131.624, -0.908, -81.97, 0.386] to (-14.06, -384.76, -8.35) mm, rotated rx 180 ry 0 rz 0 deg; joints [-0.904, -48.775, 131.589, -0.917, -81.946, 0.387]
  MoveL 1429 to (-39.46, -384.76, -8.35) mm, rotated rx -180 ry 0 rz 0 deg; joints [-0.884, -48.136, 129.627, -0.9, -80.623, 0.406]
  MoveC 1430 to (-52.16, -397.46, -8.35) mm, rotated rx 180 ry 0 rz 0 deg; joints [-1.484, -47.794, 128.617, -1.511, -79.957, 0.513] to (-64.86, -384.76, -8.35) mm, rotated rx 180 ry 0 rz 0 deg; joints [-0.865, -47.467, 127.644, -0.885, -79.309, 0.423]
  MoveL 1431 to (-90.26, -384.76, -8.35) mm, rotated rx 180 ry 0 rz 0 deg; joints [-0.847, -46.769, 125.638, -0.871, -78.001, 0.44]
  MoveL 1432 to (-166.46, -384.76, -8.35) mm, rotated rx -180 ry 0 rz 0 deg; joints [-0.798, -44.509, 119.471, -0.834, -74.094, 0.489]
  MoveC 1433 to (-179.16, -397.46, -8.35) mm, rotated rx -180 ry 0 rz 0 deg; joints [-1.341, -44.097, 118.399, -1.403, -73.437, 0.652] to (-191.86, -384.76, -8.35) mm, rotated rx 180 ry 0 rz 0 deg; joints [-0.783, -43.701, 117.361, -0.824, -72.792, 0.504]
  MoveL 1434 to (-293.46, -384.76, -8.35) mm, rotated rx -180 ry 0 rz 0 deg; joints [-0.727, -40.201, 108.598, -0.791, -67.529, 0.564]
  MoveC 1435 to (-306.16, -397.46, -8.35) mm, rotated rx -180 ry 0 rz 0 deg; joints [-1.223, -39.721, 107.442, -1.334, -66.856, 0.778] to (-318.86, -384.76, -8.35) mm, rotated rx -180 ry 0 rz 0 deg; joints [-0.714, -39.257, 106.315, -0.785, -66.191, 0.578]
  MoveL 1436 to (-395.06, -384.76, -8.35) mm, rotated rx -180 ry 0 rz 0 deg; joints [-0.679, -36.242, 99.199, -0.773, -62.09, 0.624]
  MoveL 1437 to (-420.46, -384.76, -8.35) mm, rotated rx -180 ry 0 rz 0 deg; joints [-0.668, -35.172, 96.725, -0.77, -60.685, 0.639]
  MoveC 1438 to (-433.16, -397.46, -8.35) mm, rotated rx -180 ry 0 rz 0 deg; joints [-1.124, -34.613, 95.446, -1.303, -59.97, 0.907] to (-445.86, -384.76, -8.35) mm, rotated rx -180 ry 0 rz 0 deg; joints [-0.657, -34.067, 94.192, -0.769, -59.258, 0.655]
  MoveL 1439 to (-471.26, -384.76, -8.35) mm, rotated rx -180 ry 0 rz 0 deg; joints [-0.646, -32.924, 91.595, -0.769, -57.804, 0.672]
  MoveL 1440 to (-471.26, -537.16, -8.35) mm, rotated rx -180 ry 0 rz 0 deg; joints [-6.035, -32.484, 90.662, -7.165, -57.507, 4.044]
  MoveL 1441 to (-14.06, -537.16, -8.35) mm, rotated rx -180 ry 0 rz 0 deg; joints [-8.394, -48.427, 130.628, -8.493, -81.416, 1.421]
  MoveL 1442 to (-14.06, -384.76, -8.35) mm, rotated rx 180 ry 0 rz 0 deg; joints [-0.904, -48.775, 131.589, -0.917, -81.946, 0.387]
  MoveC 1443 to (-13.87, -384.31, -8.35) mm, rotated rx 180 ry 0 rz 0 deg; joints [-0.881, -48.779, 131.604, -0.894, -81.956, 0.384] to (-13.42, -384.12, -8.35) mm, rotated rx -180 ry 0 rz 0 deg; joints [-0.873, -48.791, 131.639, -0.885, -81.98, 0.383]
  MoveL 1444 to (-12.79, -384.12, -8.35) mm, rotated rx -180 ry 0 rz 0 deg; joints [-0.873, -48.806, 131.688, -0.886, -82.013, 0.382]
  MoveC 1445 to (-12.34, -384.12, -8.16) mm, rotated rx -180 ry 0 rz 0 deg; joints [-0.873, -48.831, 131.725, -0.886, -82.025, 0.382] to (-12.15, -384.12, -7.72) mm, rotated rx -180 ry 0 rz 0 deg; joints [-0.874, -48.87, 131.745, -0.886, -82.007, 0.382]
  Set speed (1000.0 mm/s)
  MoveL 1446 to (-12.15, -384.12, 6) mm, rotated rx -180 ry 0 rz 0 deg; joints [-0.877, -49.901, 131.923, -0.891, -81.153, 0.396]
  MoveL 1447 to (-52.79, 196.51, 6) mm, rotated rx -180 ry 0 rz 0 deg; joints [25.218, -45.333, 118.689, 26.286, -74.119, -7.015]
  Set speed (25.4 mm/s)
  MoveL 1448 to (-52.79, 196.52, -4.37) mm, rotated rx -180 ry 0 rz 0 deg; joints [25.223, -44.676, 118.571, 26.224, -74.603, -6.769]
  MoveC 1449 to (-52.79, 196.7, -4.81) mm, rotated rx -180 ry 0 rz 0 deg; joints [25.23, -44.645, 118.559, 26.229, -74.621, -6.763] to (-52.79, 197.15, -5) mm, rotated rx -180 ry 0 rz 0 deg; joints [25.248, -44.628, 118.541, 26.248, -74.622, -6.767]
  Set speed (50.8 mm/s)
  MoveL 1450 to (-52.79, 197.78, -5) mm, rotated rx 180 ry 0 rz 0 deg; joints [25.273, -44.619, 118.519, 26.275, -74.613, -6.78]
  MoveC 1451 to (-52.61, 198.23, -5) mm, rotated rx 180 ry 0 rz 0 deg; joints [25.294, -44.619, 118.517, 26.297, -74.614, -6.786] to (-52.16, 198.42, -5) mm, rotated rx 180 ry 0 rz 0 deg; joints [25.309, -44.63, 118.544, 26.311, -74.631, -6.783]
  MoveL 1452 to (-14.06, 198.42, -5) mm, rotated rx -180 ry 0 rz 0 deg; joints [26.034, -45.717, 121.373, 26.852, -76.273, -6.153]
  MoveL 1453 to (-14.06, 350.82, -5) mm, rotated rx -180 ry 0 rz 0 deg; joints [31.809, -43.442, 115.252, 33.29, -73.758, -9.595]
  MoveL 1454 to (-39.46, 350.82, -5) mm, rotated rx 180 ry 0 rz 0 deg; joints [31.254, -42.694, 113.399, 32.901, -72.736, -10.069]
  MoveC 1455 to (-52.16, 338.12, -5) mm, rotated rx -180 ry 0 rz 0 deg; joints [30.534, -42.53, 113.02, 32.194, -72.425, -9.979] to (-64.86, 350.82, -5) mm, rotated rx 180 ry 0 rz 0 deg; joints [30.717, -41.922, 111.511, 32.54, -71.698, -10.541]
  MoveL 1456 to (-90.26, 350.82, -5) mm, rotated rx -180 ry 0 rz 0 deg; joints [30.196, -41.126, 109.586, 32.206, -70.645, -11.013]
  MoveL 1457 to (-166.46, 350.82, -5) mm, rotated rx 180 ry 0 rz 0 deg; joints [28.725, -38.589, 103.572, 31.367, -67.383, -12.445]
  MoveC 1458 to (-179.16, 338.12, -5) mm, rotated rx -180 ry 0 rz 0 deg; joints [28.065, -38.375, 103.092, 30.726, -67.011, -12.333] to (-191.86, 350.82, -5) mm, rotated rx -180 ry 0 rz 0 deg; joints [28.263, -37.69, 101.48, 31.142, -66.26, -12.933]
  MoveL 1459 to (-293.46, 350.82, -5) mm, rotated rx 180 ry 0 rz 0 deg; joints [26.546, -33.799, 92.606, 30.539, -61.558, -14.988]
  MoveC 1460 to (-306.16, 338.12, -5) mm, rotated rx -180 ry 0 rz 0 deg; joints [25.94, -33.526, 92.009, 29.962, -61.119, -14.864] to (-318.86, 350.82, -5) mm, rotated rx -180 ry 0 rz 0 deg; joints [26.146, -32.743, 90.241, 30.469, -60.323, -15.541]
  MoveL 1461 to (-395.06, 350.82, -5) mm, rotated rx -180 ry 0 rz 0 deg; joints [25.013, -29.34, 82.711, 30.482, -56.44, -17.347]
  MoveL 1462 to (-420.46, 350.82, -5) mm, rotated rx -180 ry 0 rz 0 deg; joints [24.655, -28.115, 80.031, 30.573, -55.077, -18.014]
  MoveC 1463 to (-433.16, 338.12, -5) mm, rotated rx 180 ry 0 rz 0 deg; joints [24.096, -27.763, 79.278, 30.066, -54.555, -17.896] to (-445.86, 350.82, -5) mm, rotated rx -180 ry 0 rz 0 deg; joints [24.307, -26.836, 77.25, 30.716, -53.673, -18.725]
  MoveL 1464 to (-471.26, 350.82, -5) mm, rotated rx -180 ry 0 rz 0 deg; joints [23.968, -25.498, 74.355, 30.917, -52.223, -19.488]
  MoveL 1465 to (-471.26, 198.42, -5) mm, rotated rx -180 ry 0 rz 0 deg; joints [19.296, -28.569, 81.175, 24.04, -54.184, -14.052]
  MoveL 1466 to (-445.86, 198.42, -5) mm, rotated rx -180 ry 0 rz 0 deg; joints [19.581, -29.819, 83.919, 23.95, -55.619, -13.5]
  MoveL 1467 to (-52.16, 198.42, -5) mm, rotated rx -180 ry 0 rz 0 deg; joints [25.309, -44.63, 118.544, 26.311, -74.631, -6.783]
  MoveC 1468 to (-51.71, 198.23, -5) mm, rotated rx -180 ry 0 rz 0 deg; joints [25.31, -44.645, 118.584, 26.309, -74.653, -6.772] to (-51.52, 197.78, -5) mm, rotated rx 180 ry 0 rz 0 deg; joints [25.296, -44.656, 118.614, 26.292, -74.668, -6.76]
  MoveL 1469 to (-51.52, 197.15, -5) mm, rotated rx 180 ry 0 rz 0 deg; joints [25.271, -44.665, 118.637, 26.265, -74.678, -6.747]
  MoveC 1470 to (-51.52, 196.7, -4.81) mm, rotated rx 180 ry 0 rz 0 deg; joints [25.254, -44.682, 118.655, 26.246, -74.676, -6.742] to (-51.52, 196.52, -4.37) mm, rotated rx -180 ry 0 rz 0 deg; joints [25.246, -44.713, 118.667, 26.241, -74.658, -6.749]
  Set speed (1000.0 mm/s)
  MoveL 1471 to (-51.52, 196.51, 5) mm, rotated rx 180 ry 0 rz 0 deg; joints [25.242, -45.307, 118.774, 26.297, -74.221, -6.971]
  MoveL 1472 to (-52.79, 196.51, 5) mm, rotated rx -180 ry 0 rz 0 deg; joints [25.218, -45.269, 118.678, 26.28, -74.166, -6.991]
  Set speed (25.4 mm/s)
  MoveL 1473 to (-52.79, 196.52, 1) mm, rotated rx -180 ry 0 rz 0 deg; joints [25.22, -45.016, 118.633, 26.255, -74.353, -6.896]
  MoveL 1474 to (-52.79, 196.52, -7.71) mm, rotated rx -180 ry 0 rz 0 deg; joints [25.224, -44.463, 118.531, 26.205, -74.758, -6.691]
  MoveC 1475 to (-52.79, 196.7, -8.16) mm, rotated rx 180 ry 0 rz 0 deg; joints [25.232, -44.433, 118.519, 26.21, -74.776, -6.684] to (-52.79, 197.15, -8.35) mm, rotated rx -180 ry 0 rz 0 deg; joints [25.249, -44.415, 118.501, 26.228, -74.777, -6.689]
  Set speed (50.8 mm/s)
  MoveL 1476 to (-52.79, 197.78, -8.35) mm, rotated rx -180 ry 0 rz 0 deg; joints [25.274, -44.407, 118.478, 26.256, -74.768, -6.702]
  MoveC 1477 to (-52.61, 198.23, -8.35) mm, rotated rx -180 ry 0 rz 0 deg; joints [25.295, -44.406, 118.477, 26.278, -74.769, -6.708] to (-52.16, 198.42, -8.35) mm, rotated rx 180 ry 0 rz 0 deg; joints [25.311, -44.417, 118.504, 26.292, -74.785, -6.704]
  MoveL 1478 to (-14.06, 198.42, -8.35) mm, rotated rx -180 ry 0 rz 0 deg; joints [26.036, -45.497, 121.332, 26.834, -76.433, -6.071]
  MoveL 1479 to (-14.06, 350.82, -8.35) mm, rotated rx -180 ry 0 rz 0 deg; joints [31.811, -43.237, 115.212, 33.265, -73.897, -9.501]
  MoveL 1480 to (-39.46, 350.82, -8.35) mm, rotated rx -180 ry 0 rz 0 deg; joints [31.256, -42.493, 113.36, 32.875, -72.872, -9.977]
  MoveC 1481 to (-52.16, 338.12, -8.35) mm, rotated rx -180 ry 0 rz 0 deg; joints [30.535, -42.329, 112.98, 32.169, -72.562, -9.889] to (-64.86, 350.82, -8.35) mm, rotated rx 180 ry 0 rz 0 deg; joints [30.718, -41.725, 111.472, 32.513, -71.832, -10.452]
  MoveL 1482 to (-90.26, 350.82, -8.35) mm, rotated rx -180 ry 0 rz 0 deg; joints [30.197, -40.932, 109.547, 32.178, -70.776, -10.926]
  MoveL 1483 to (-166.46, 350.82, -8.35) mm, rotated rx -180 ry 0 rz 0 deg; joints [28.726, -38.405, 103.534, 31.337, -67.508, -12.363]
  MoveC 1484 to (-179.16, 338.12, -8.35) mm, rotated rx -180 ry 0 rz 0 deg; joints [28.067, -38.192, 103.054, 30.697, -67.136, -12.253] to (-191.86, 350.82, -8.35) mm, rotated rx 180 ry 0 rz 0 deg; joints [28.265, -37.509, 101.442, 31.111, -66.382, -12.853]
  MoveL 1485 to (-293.46, 350.82, -8.35) mm, rotated rx 180 ry 0 rz 0 deg; joints [26.547, -33.629, 92.567, 30.505, -61.671, -14.913]
  MoveC 1486 to (-306.16, 338.12, -8.35) mm, rotated rx -180 ry 0 rz 0 deg; joints [25.941, -33.357, 91.97, 29.928, -61.233, -14.79] to (-318.86, 350.82, -8.35) mm, rotated rx -180 ry 0 rz 0 deg; joints [26.148, -32.576, 90.202, 30.433, -60.434, -15.466]
  MoveL 1487 to (-395.06, 350.82, -8.35) mm, rotated rx 180 ry 0 rz 0 deg; joints [25.014, -29.18, 82.671, 30.443, -56.544, -17.274]
  MoveL 1488 to (-420.46, 350.82, -8.35) mm, rotated rx 180 ry 0 rz 0 deg; joints [24.656, -27.956, 79.99, 30.533, -55.179, -17.942]
  MoveC 1489 to (-433.16, 338.12, -8.35) mm, rotated rx -180 ry 0 rz 0 deg; joints [24.097, -27.605, 79.237, 30.026, -54.657, -17.825] to (-445.86, 350.82, -8.35) mm, rotated rx 180 ry 0 rz 0 deg; joints [24.308, -26.679, 77.209, 30.674, -53.772, -18.653]
  MoveL 1490 to (-471.26, 350.82, -8.35) mm, rotated rx -180 ry 0 rz 0 deg; joints [23.969, -25.343, 74.313, 30.874, -52.32, -19.416]
  MoveL 1491 to (-471.26, 198.42, -8.35) mm, rotated rx 180 ry 0 rz 0 deg; joints [19.297, -28.409, 81.134, 24.006, -54.293, -13.994]
  MoveL 1492 to (-445.86, 198.42, -8.35) mm, rotated rx -180 ry 0 rz 0 deg; joints [19.582, -29.657, 83.879, 23.918, -55.73, -13.441]
  MoveL 1493 to (-52.16, 198.42, -8.35) mm, rotated rx 180 ry 0 rz 0 deg; joints [25.311, -44.417, 118.504, 26.292, -74.785, -6.704]
  MoveC 1494 to (-51.71, 198.23, -8.35) mm, rotated rx -180 ry 0 rz 0 deg; joints [25.312, -44.432, 118.544, 26.29, -74.808, -6.693] to (-51.52, 197.78, -8.35) mm, rotated rx 180 ry 0 rz 0 deg; joints [25.298, -44.444, 118.574, 26.273, -74.823, -6.681]
  MoveL 1495 to (-51.52, 197.15, -8.35) mm, rotated rx 180 ry 0 rz 0 deg; joints [25.273, -44.452, 118.596, 26.246, -74.833, -6.668]
  MoveC 1496 to (-51.52, 196.7, -8.16) mm, rotated rx 180 ry 0 rz 0 deg; joints [25.255, -44.469, 118.614, 26.227, -74.831, -6.663] to (-51.52, 196.52, -7.72) mm, rotated rx -180 ry 0 rz 0 deg; joints [25.248, -44.5, 118.626, 26.222, -74.813, -6.67]
  Set speed (1000.0 mm/s)
  MoveL 1497 to (-51.52, 196.51, 6) mm, rotated rx -180 ry 0 rz 0 deg; joints [25.241, -45.37, 118.785, 26.303, -74.174, -6.995]
  MoveL 1498 to (18.41, 196.51, 6) mm, rotated rx 180 ry 0 rz 0 deg; joints [26.6, -47.366, 123.93, 27.332, -77.143, -5.853]
  Set speed (25.4 mm/s)
  MoveL 1499 to (18.41, 196.52, -4.37) mm, rotated rx -180 ry 0 rz 0 deg; joints [26.605, -46.668, 123.808, 27.279, -77.656, -5.583]
  MoveC 1500 to (18.41, 196.7, -4.81) mm, rotated rx -180 ry 0 rz 0 deg; joints [26.613, -46.635, 123.796, 27.285, -77.675, -5.575] to (18.41, 197.15, -5) mm, rotated rx -180 ry 0 rz 0 deg; joints [26.631, -46.617, 123.777, 27.303, -77.677, -5.579]
  Set speed (50.8 mm/s)
  MoveL 1501 to (18.41, 197.78, -5) mm, rotated rx 180 ry 0 rz 0 deg; joints [26.657, -46.609, 123.754, 27.331, -77.666, -5.591]
  MoveC 1502 to (18.6, 198.23, -5) mm, rotated rx -180 ry 0 rz 0 deg; joints [26.679, -46.608, 123.752, 27.354, -77.666, -5.597] to (19.05, 198.42, -5) mm, rotated rx -180 ry 0 rz 0 deg; joints [26.696, -46.618, 123.777, 27.369, -77.682, -5.592]
  MoveL 1503 to (39.46, 198.42, -5) mm, rotated rx -180 ry 0 rz 0 deg; joints [27.12, -47.153, 125.235, 27.71, -78.543, -5.239]
  MoveL 1504 to (471.26, 198.42, -5) mm, rotated rx -180 ry 0 rz 0 deg; joints [40.082, -54.215, 152.16, 40.272, -95.205, 5.399]
  MoveL 1505 to (471.26, 350.82, -5) mm, rotated rx -180 ry 0 rz 0 deg; joints [46.899, -53.296, 144.736, 46.888, -90.115, 1.324]
  MoveL 1506 to (445.86, 350.82, -5) mm, rotated rx 180 ry 0 rz 0 deg; joints [45.836, -53.001, 143.464, 45.828, -89.453, 0.604]
  MoveC 1507 to (433.16, 338.12, -5) mm, rotated rx 180 ry 0 rz 0 deg; joints [44.807, -52.979, 143.467, 44.799, -89.477, 0.616] to (420.46, 350.82, -5) mm, rotated rx 180 ry 0 rz 0 deg; joints [44.811, -52.68, 142.16, 44.813, -88.762, -0.094]
  MoveL 1508 to (395.06, 350.82, -5) mm, rotated rx 180 ry 0 rz 0 deg; joints [43.821, -52.333, 140.825, 43.842, -88.043, -0.772]
  MoveL 1509 to (318.86, 350.82, -5) mm, rotated rx -180 ry 0 rz 0 deg; joints [41.052, -51.14, 136.641, 41.181, -85.74, -2.689]
  MoveC 1510 to (306.16, 338.12, -5) mm, rotated rx -180 ry 0 rz 0 deg; joints [40.114, -51.09, 136.533, 40.244, -85.648, -2.67] to (293.46, 350.82, -5) mm, rotated rx -180 ry 0 rz 0 deg; joints [40.193, -50.693, 135.187, 40.373, -84.929, -3.291]
  MoveL 1511 to (191.86, 350.82, -5) mm, rotated rx -180 ry 0 rz 0 deg; joints [37.037, -48.668, 129.083, 37.51, -81.496, -5.547]
  MoveC 1512 to (179.16, 338.12, -5) mm, rotated rx 180 ry 0 rz 0 deg; joints [36.183, -48.581, 128.875, 36.662, -81.313, -5.506] to (166.46, 350.82, -5) mm, rotated rx 180 ry 0 rz 0 deg; joints [36.313, -48.104, 127.484, 36.88, -80.596, -6.078]
  MoveL 1513 to (90.26, 350.82, -5) mm, rotated rx -180 ry 0 rz 0 deg; joints [34.283, -46.275, 122.512, 35.181, -77.801, -7.607]
  MoveL 1514 to (64.86, 350.82, -5) mm, rotated rx -180 ry 0 rz 0 deg; joints [33.65, -45.62, 120.793, 34.676, -76.84, -8.1]
  MoveC 1515 to (61.14, 341.84, -5) mm, rotated rx -180 ry 0 rz 0 deg; joints [33.227, -45.67, 120.943, 34.233, -76.861, -7.951] to (52.16, 338.12, -5) mm, rotated rx -180 ry 0 rz 0 deg; joints [32.873, -45.493, 120.491, 33.909, -76.583, -8.032]
  MoveL 1516 to (52.16, 338.12, -5) mm, rotated rx -180 ry 0 rz 0 deg; joints [32.873, -45.493, 120.491, 33.909, -76.583, -8.032]
  MoveC 1517 to (43.18, 341.84, -5) mm, rotated rx -180 ry 0 rz 0 deg; joints [32.796, -45.192, 119.704, 33.897, -76.168, -8.293] to (39.46, 350.82, -5) mm, rotated rx -180 ry 0 rz 0 deg; joints [33.037, -44.943, 119.044, 34.2, -75.863, -8.586]
  MoveL 1518 to (14.06, 350.82, -5) mm, rotated rx 180 ry 0 rz 0 deg; joints [32.444, -44.243, 117.262, 33.752, -74.872, -9.067]
  MoveL 1519 to (14.06, 198.42, -5) mm, rotated rx 180 ry 0 rz 0 deg; joints [26.594, -46.485, 123.418, 27.288, -77.471, -5.678]
  MoveL 1520 to (19.05, 198.42, -5) mm, rotated rx -180 ry 0 rz 0 deg; joints [26.696, -46.618, 123.777, 27.369, -77.682, -5.592]
  MoveC 1521 to (19.49, 198.23, -5) mm, rotated rx -180 ry 0 rz 0 deg; joints [26.698, -46.632, 123.816, 27.368, -77.704, -5.581] to (19.68, 197.78, -5) mm, rotated rx -180 ry 0 rz 0 deg; joints [26.683, -46.643, 123.846, 27.352, -77.72, -5.569]
  MoveL 1522 to (19.68, 197.15, -5) mm, rotated rx 180 ry 0 rz 0 deg; joints [26.657, -46.651, 123.868, 27.324, -77.73, -5.557]
  MoveC 1523 to (19.68, 196.7, -4.81) mm, rotated rx 180 ry 0 rz 0 deg; joints [26.639, -46.669, 123.887, 27.305, -77.729, -5.553] to (19.68, 196.52, -4.37) mm, rotated rx -180 ry 0 rz 0 deg; joints [26.631, -46.702, 123.899, 27.299, -77.71, -5.561]
  Set speed (1000.0 mm/s)
  MoveL 1524 to (19.68, 196.52, 5) mm, rotated rx -180 ry 0 rz 0 deg; joints [26.626, -47.334, 124.01, 27.348, -77.246, -5.805]
  MoveL 1525 to (18.41, 196.51, 5) mm, rotated rx -180 ry 0 rz 0 deg; joints [26.6, -47.299, 123.919, 27.327, -77.193, -5.827]
  Set speed (25.4 mm/s)
  MoveL 1526 to (18.41, 196.51, 1) mm, rotated rx -180 ry 0 rz 0 deg; joints [26.602, -47.03, 123.872, 27.306, -77.391, -5.722]
  MoveL 1527 to (18.41, 196.51, -7.71) mm, rotated rx -180 ry 0 rz 0 deg; joints [26.607, -46.441, 123.766, 27.262, -77.82, -5.497]
  MoveC 1528 to (18.41, 196.7, -8.16) mm, rotated rx -180 ry 0 rz 0 deg; joints [26.615, -46.409, 123.754, 27.268, -77.839, -5.489] to (18.41, 197.15, -8.35) mm, rotated rx -180 ry 0 rz 0 deg; joints [26.633, -46.391, 123.735, 27.287, -77.841, -5.493]
  Set speed (50.8 mm/s)
  MoveL 1529 to (18.41, 197.78, -8.35) mm, rotated rx -180 ry 0 rz 0 deg; joints [26.659, -46.383, 123.713, 27.314, -77.83, -5.505]
  MoveC 1530 to (18.6, 198.23, -8.35) mm, rotated rx -180 ry 0 rz 0 deg; joints [26.681, -46.382, 123.71, 27.337, -77.83, -5.51] to (19.04, 198.42, -8.35) mm, rotated rx -180 ry 0 rz 0 deg; joints [26.698, -46.392, 123.735, 27.353, -77.846, -5.506]
  MoveL 1531 to (39.46, 198.42, -8.35) mm, rotated rx -180 ry 0 rz 0 deg; joints [27.122, -46.922, 125.193, 27.694, -78.71, -5.15]
  MoveL 1532 to (471.26, 198.42, -8.35) mm, rotated rx -180 ry 0 rz 0 deg; joints [40.085, -53.848, 152.098, 40.294, -95.438, 5.598]
  MoveL 1533 to (471.26, 350.82, -8.35) mm, rotated rx -180 ry 0 rz 0 deg; joints [46.902, -52.982, 144.683, 46.891, -90.293, 1.514]
  MoveL 1534 to (445.86, 350.82, -8.35) mm, rotated rx 180 ry 0 rz 0 deg; joints [45.839, -52.695, 143.412, 45.829, -89.63, 0.787]
  MoveC 1535 to (433.16, 338.12, -8.35) mm, rotated rx 180 ry 0 rz 0 deg; joints [44.81, -52.673, 143.415, 44.8, -89.657, 0.795] to (420.46, 350.82, -8.35) mm, rotated rx 180 ry 0 rz 0 deg; joints [44.813, -52.381, 142.109, 44.812, -88.938, 0.081]
  MoveL 1536 to (395.06, 350.82, -8.35) mm, rotated rx 180 ry 0 rz 0 deg; joints [43.823, -52.041, 140.775, 43.839, -88.218, -0.604]
  MoveL 1537 to (318.86, 350.82, -8.35) mm, rotated rx -180 ry 0 rz 0 deg; joints [41.055, -50.868, 136.594, 41.172, -85.909, -2.54]
  MoveC 1538 to (306.16, 338.12, -8.35) mm, rotated rx -180 ry 0 rz 0 deg; joints [40.116, -50.819, 136.486, 40.235, -85.819, -2.525] to (293.46, 350.82, -8.35) mm, rotated rx -180 ry 0 rz 0 deg; joints [40.195, -50.427, 135.141, 40.363, -85.096, -3.149]
  MoveL 1539 to (191.86, 350.82, -8.35) mm, rotated rx -180 ry 0 rz 0 deg; joints [37.039, -48.425, 129.039, 37.494, -81.655, -5.425]
  MoveC 1540 to (179.16, 338.12, -8.35) mm, rotated rx -180 ry 0 rz 0 deg; joints [36.185, -48.339, 128.832, 36.646, -81.473, -5.386] to (166.46, 350.82, -8.35) mm, rotated rx -180 ry 0 rz 0 deg; joints [36.315, -47.866, 127.441, 36.863, -80.752, -5.96]
  MoveL 1541 to (90.26, 350.82, -8.35) mm, rotated rx -180 ry 0 rz 0 deg; joints [34.285, -46.052, 122.47, 35.161, -77.95, -7.501]
  MoveL 1542 to (64.86, 350.82, -8.35) mm, rotated rx 180 ry 0 rz 0 deg; joints [33.652, -45.402, 120.753, 34.654, -76.986, -7.997]
  MoveC 1543 to (61.14, 341.84, -8.35) mm, rotated rx -180 ry 0 rz 0 deg; joints [33.229, -45.451, 120.902, 34.212, -77.009, -7.848] to (52.16, 338.12, -8.35) mm, rotated rx 180 ry 0 rz 0 deg; joints [32.875, -45.275, 120.451, 33.888, -76.73, -7.931]
  MoveL 1544 to (52.16, 338.12, -8.35) mm, rotated rx 180 ry 0 rz 0 deg; joints [32.875, -45.275, 120.451, 33.888, -76.73, -7.931]
  MoveC 1545 to (43.18, 341.84, -8.35) mm, rotated rx -180 ry 0 rz 0 deg; joints [32.798, -44.977, 119.664, 33.875, -76.313, -8.193] to (39.46, 350.82, -8.35) mm, rotated rx -180 ry 0 rz 0 deg; joints [33.039, -44.729, 119.004, 34.177, -76.007, -8.486]
  MoveL 1546 to (14.06, 350.82, -8.35) mm, rotated rx -180 ry 0 rz 0 deg; joints [32.446, -44.034, 117.222, 33.729, -75.014, -8.97]
  MoveL 1547 to (14.06, 198.42, -8.35) mm, rotated rx 180 ry 0 rz 0 deg; joints [26.596, -46.259, 123.376, 27.272, -77.634, -5.592]
  MoveL 1548 to (19.04, 198.42, -8.35) mm, rotated rx -180 ry 0 rz 0 deg; joints [26.698, -46.392, 123.735, 27.353, -77.846, -5.506]
  MoveC 1549 to (19.49, 198.23, -8.35) mm, rotated rx -180 ry 0 rz 0 deg; joints [26.699, -46.406, 123.774, 27.352, -77.869, -5.495] to (19.68, 197.78, -8.35) mm, rotated rx 180 ry 0 rz 0 deg; joints [26.685, -46.416, 123.804, 27.335, -77.884, -5.483]
  MoveL 1550 to (19.68, 197.15, -8.35) mm, rotated rx -180 ry 0 rz 0 deg; joints [26.659, -46.424, 123.827, 27.307, -77.895, -5.471]
  MoveC 1551 to (19.68, 196.7, -8.16) mm, rotated rx -180 ry 0 rz 0 deg; joints [26.641, -46.442, 123.845, 27.289, -77.893, -5.467] to (19.68, 196.52, -7.72) mm, rotated rx -180 ry 0 rz 0 deg; joints [26.633, -46.475, 123.857, 27.283, -77.874, -5.475]
  Set speed (1000.0 mm/s)
  MoveL 1552 to (19.68, 196.51, 6) mm, rotated rx -180 ry 0 rz 0 deg; joints [26.626, -47.401, 124.021, 27.353, -77.196, -5.832]
  MoveL 1553 to (18.41, 382.85, 6) mm, rotated rx 180 ry 0 rz 0 deg; joints [33.684, -44.487, 116.227, 35.222, -74.03, -10.14]
  Set speed (25.4 mm/s)
  MoveL 1554 to (18.41, 382.85, -4.36) mm, rotated rx -180 ry 0 rz 0 deg; joints [33.689, -43.849, 116.111, 35.142, -74.458, -9.829]
  MoveC 1555 to (18.41, 383.04, -4.81) mm, rotated rx -180 ry 0 rz 0 deg; joints [33.696, -43.818, 116.097, 35.147, -74.474, -9.82] to (18.41, 383.49, -5) mm, rotated rx -180 ry 0 rz 0 deg; joints [33.712, -43.798, 116.074, 35.164, -74.473, -9.827]
  Set speed (50.8 mm/s)
  MoveL 1556 to (18.41, 384.12, -5) mm, rotated rx -180 ry 0 rz 0 deg; joints [33.734, -43.787, 116.044, 35.189, -74.462, -9.844]
  MoveC 1557 to (18.6, 384.57, -5) mm, rotated rx -180 ry 0 rz 0 deg; joints [33.755, -43.784, 116.036, 35.211, -74.462, -9.852] to (19.04, 384.76, -5) mm, rotated rx -180 ry 0 rz 0 deg; joints [33.772, -43.794, 116.059, 35.226, -74.476, -9.848]
  MoveL 1558 to (64.86, 384.76, -5) mm, rotated rx -180 ry 0 rz 0 deg; joints [34.882, -45.044, 119.225, 36.066, -76.219, -8.964]
  MoveL 1559 to (471.26, 384.76, -5) mm, rotated rx -180 ry 0 rz 0 deg; joints [48.218, -52.932, 142.927, 48.214, -89.127, 0.268]
  MoveL 1560 to (471.26, 537.16, -5) mm, rotated rx -180 ry 0 rz 0 deg; joints [53.393, -50.654, 134.164, 53.645, -85.269, -4.951]
  MoveL 1561 to (445.86, 537.16, -5) mm, rotated rx -180 ry 0 rz 0 deg; joints [52.37, -50.264, 132.993, 52.677, -84.703, -5.505]
  MoveC 1562 to (433.16, 524.46, -5) mm, rotated rx -180 ry 0 rz 0 deg; joints [51.474, -50.296, 133.154, 51.772, -84.693, -5.333] to (420.46, 537.16, -5) mm, rotated rx -180 ry 0 rz 0 deg; joints [51.373, -49.854, 131.787, 51.743, -84.11, -6.055]
  MoveL 1563 to (395.06, 537.16, -5) mm, rotated rx 180 ry 0 rz 0 deg; joints [50.404, -49.425, 130.547, 50.843, -83.491, -6.601]
  MoveL 1564 to (318.86, 537.16, -5) mm, rotated rx -180 ry 0 rz 0 deg; joints [47.652, -48.019, 126.627, 48.344, -81.493, -8.216]
  MoveC 1565 to (306.16, 524.46, -5) mm, rotated rx -180 ry 0 rz 0 deg; joints [46.811, -48.021, 126.679, 47.497, -81.404, -8.065] to (293.46, 537.16, -5) mm, rotated rx -180 ry 0 rz 0 deg; joints [46.785, -47.511, 125.254, 47.577, -80.781, -8.745]
  MoveL 1566 to (191.86, 537.16, -5) mm, rotated rx -180 ry 0 rz 0 deg; joints [43.549, -45.278, 119.427, 44.825, -77.728, -10.83]
  MoveC 1567 to (179.16, 524.46, -5) mm, rotated rx -180 ry 0 rz 0 deg; joints [42.765, -45.244, 119.376, 44.04, -77.566, -10.686] to (166.46, 537.16, -5) mm, rotated rx -180 ry 0 rz 0 deg; joints [42.795, -44.669, 117.886, 44.215, -76.915, -11.345]
  MoveL 1568 to (90.26, 537.16, -5) mm, rotated rx -180 ry 0 rz 0 deg; joints [40.656, -42.715, 113.053, 42.565, -74.364, -12.885]
  MoveL 1569 to (64.86, 537.16, -5) mm, rotated rx 180 ry 0 rz 0 deg; joints [39.982, -42.02, 111.37, 42.074, -73.476, -13.399]
  MoveC 1570 to (61.14, 528.18, -5) mm, rotated rx -180 ry 0 rz 0 deg; joints [39.604, -42.116, 111.62, 41.66, -73.503, -13.187] to (52.16, 524.46, -5) mm, rotated rx -180 ry 0 rz 0 deg; joints [39.254, -41.946, 111.22, 41.351, -73.248, -13.251]
  MoveL 1571 to (52.16, 524.46, -5) mm, rotated rx -180 ry 0 rz 0 deg; joints [39.254, -41.946, 111.22, 41.351, -73.248, -13.251]
  MoveC 1572 to (43.18, 528.18, -5) mm, rotated rx 180 ry 0 rz 0 deg; joints [39.141, -41.61, 110.403, 41.333, -72.861, -13.551] to (39.46, 537.16, -5) mm, rotated rx -180 ry 0 rz 0 deg; joints [39.327, -41.304, 109.649, 41.614, -72.57, -13.915]
  MoveL 1573 to (14.06, 537.16, -5) mm, rotated rx 180 ry 0 rz 0 deg; joints [38.689, -40.564, 107.889, 41.182, -71.646, -14.434]
  MoveL 1574 to (14.06, 384.76, -5) mm, rotated rx -180 ry 0 rz 0 deg; joints [33.655, -43.653, 115.708, 35.14, -74.283, -9.944]
  MoveL 1575 to (19.04, 384.76, -5) mm, rotated rx -180 ry 0 rz 0 deg; joints [33.772, -43.794, 116.059, 35.226, -74.476, -9.848]
  MoveC 1576 to (19.49, 384.57, -5) mm, rotated rx 180 ry 0 rz 0 deg; joints [33.776, -43.809, 116.099, 35.226, -74.496, -9.835] to (19.68, 384.12, -5) mm, rotated rx -180 ry 0 rz 0 deg; joints [33.764, -43.823, 116.133, 35.211, -74.511, -9.819]
  MoveL 1577 to (19.68, 383.49, -5) mm, rotated rx 180 ry 0 rz 0 deg; joints [33.742, -43.834, 116.163, 35.186, -74.523, -9.802]
  MoveC 1578 to (19.68, 383.04, -4.81) mm, rotated rx 180 ry 0 rz 0 deg; joints [33.726, -43.854, 116.186, 35.169, -74.523, -9.796] to (19.68, 382.85, -4.37) mm, rotated rx -180 ry 0 rz 0 deg; joints [33.719, -43.885, 116.2, 35.164, -74.508, -9.805]
  Set speed (1000.0 mm/s)
  MoveL 1579 to (19.68, 382.85, 5) mm, rotated rx -180 ry 0 rz 0 deg; joints [33.714, -44.462, 116.305, 35.236, -74.121, -10.086]
  MoveL 1580 to (18.41, 382.85, 5) mm, rotated rx -180 ry 0 rz 0 deg; joints [33.684, -44.426, 116.216, 35.214, -74.072, -10.11]
  Set speed (25.4 mm/s)
  MoveL 1581 to (18.41, 382.85, 1) mm, rotated rx 180 ry 0 rz 0 deg; joints [33.686, -44.18, 116.172, 35.183, -74.237, -9.99]
  MoveL 1582 to (18.41, 382.85, -7.71) mm, rotated rx -180 ry 0 rz 0 deg; joints [33.691, -43.642, 116.071, 35.118, -74.596, -9.729]
  MoveC 1583 to (18.41, 383.04, -8.16) mm, rotated rx 180 ry 0 rz 0 deg; joints [33.698, -43.611, 116.057, 35.122, -74.611, -9.721] to (18.41, 383.49, -8.35) mm, rotated rx -180 ry 0 rz 0 deg; joints [33.714, -43.591, 116.034, 35.139, -74.611, -9.727]
  Set speed (50.8 mm/s)
  MoveL 1584 to (18.41, 384.12, -8.35) mm, rotated rx -180 ry 0 rz 0 deg; joints [33.736, -43.58, 116.005, 35.164, -74.599, -9.744]
  MoveC 1585 to (18.6, 384.57, -8.35) mm, rotated rx -180 ry 0 rz 0 deg; joints [33.756, -43.577, 115.997, 35.186, -74.599, -9.752] to (19.04, 384.76, -8.35) mm, rotated rx -180 ry 0 rz 0 deg; joints [33.774, -43.587, 116.019, 35.201, -74.613, -9.749]
  MoveL 1586 to (64.86, 384.76, -8.35) mm, rotated rx -180 ry 0 rz 0 deg; joints [34.884, -44.83, 119.185, 36.043, -76.36, -8.859]
  MoveL 1587 to (471.26, 384.76, -8.35) mm, rotated rx -180 ry 0 rz 0 deg; joints [48.221, -52.629, 142.875, 48.214, -89.294, 0.456]
  MoveL 1588 to (471.26, 537.16, -8.35) mm, rotated rx -180 ry 0 rz 0 deg; joints [53.396, -50.393, 134.119, 53.633, -85.397, -4.777]
  MoveL 1589 to (445.86, 537.16, -8.35) mm, rotated rx 180 ry 0 rz 0 deg; joints [52.372, -50.007, 132.948, 52.664, -84.831, -5.336]
  MoveC 1590 to (433.16, 524.46, -8.35) mm, rotated rx -180 ry 0 rz 0 deg; joints [51.476, -50.039, 133.109, 51.759, -84.825, -5.165] to (420.46, 537.16, -8.35) mm, rotated rx -180 ry 0 rz 0 deg; joints [51.376, -49.602, 131.743, 51.729, -84.239, -5.891]
  MoveL 1591 to (395.06, 537.16, -8.35) mm, rotated rx 180 ry 0 rz 0 deg; joints [50.406, -49.177, 130.503, 50.828, -83.62, -6.442]
  MoveL 1592 to (318.86, 537.16, -8.35) mm, rotated rx -180 ry 0 rz 0 deg; joints [47.654, -47.785, 126.585, 48.325, -81.621, -8.071]
  MoveC 1593 to (306.16, 524.46, -8.35) mm, rotated rx -180 ry 0 rz 0 deg; joints [46.813, -47.786, 126.637, 47.478, -81.534, -7.922] to (293.46, 537.16, -8.35) mm, rotated rx -180 ry 0 rz 0 deg; joints [46.787, -47.281, 125.212, 47.557, -80.909, -8.605]
  MoveL 1594 to (191.86, 537.16, -8.35) mm, rotated rx 180 ry 0 rz 0 deg; joints [43.551, -45.063, 119.387, 44.801, -77.852, -10.705]
  MoveC 1595 to (179.16, 524.46, -8.35) mm, rotated rx -180 ry 0 rz 0 deg; joints [42.767, -45.029, 119.336, 44.016, -77.692, -10.562] to (166.46, 537.16, -8.35) mm, rotated rx -180 ry 0 rz 0 deg; joints [42.797, -44.458, 117.846, 44.189, -77.038, -11.223]
  MoveL 1596 to (90.26, 537.16, -8.35) mm, rotated rx -180 ry 0 rz 0 deg; joints [40.658, -42.514, 113.014, 42.536, -74.483, -12.772]
  MoveL 1597 to (64.86, 537.16, -8.35) mm, rotated rx 180 ry 0 rz 0 deg; joints [39.984, -41.823, 111.331, 42.045, -73.594, -13.289]
  MoveC 1598 to (61.14, 528.18, -8.35) mm, rotated rx 180 ry 0 rz 0 deg; joints [39.606, -41.918, 111.582, 41.631, -73.622, -13.078] to (52.16, 524.46, -8.35) mm, rotated rx -180 ry 0 rz 0 deg; joints [39.256, -41.749, 111.181, 41.322, -73.368, -13.142]
  MoveL 1599 to (52.16, 524.46, -8.35) mm, rotated rx 180 ry 0 rz 0 deg; joints [39.256, -41.749, 111.181, 41.322, -73.368, -13.142]
  MoveC 1600 to (43.18, 528.18, -8.35) mm, rotated rx -180 ry 0 rz 0 deg; joints [39.143, -41.415, 110.365, 41.303, -72.979, -13.443] to (39.46, 537.16, -8.35) mm, rotated rx -180 ry 0 rz 0 deg; joints [39.328, -41.11, 109.61, 41.583, -72.687, -13.807]
  MoveL 1601 to (14.06, 537.16, -8.35) mm, rotated rx -180 ry 0 rz 0 deg; joints [38.691, -40.374, 107.851, 41.151, -71.761, -14.329]
  MoveL 1602 to (14.06, 384.76, -8.35) mm, rotated rx 180 ry 0 rz 0 deg; joints [33.656, -43.447, 115.668, 35.115, -74.419, -9.845]
  MoveL 1603 to (19.04, 384.76, -8.35) mm, rotated rx -180 ry 0 rz 0 deg; joints [33.774, -43.587, 116.019, 35.201, -74.613, -9.749]
  MoveC 1604 to (19.49, 384.57, -8.35) mm, rotated rx -180 ry 0 rz 0 deg; joints [33.778, -43.602, 116.06, 35.201, -74.634, -9.735] to (19.68, 384.12, -8.35) mm, rotated rx -180 ry 0 rz 0 deg; joints [33.766, -43.616, 116.094, 35.186, -74.649, -9.72]
  MoveL 1605 to (19.68, 383.49, -8.35) mm, rotated rx 180 ry 0 rz 0 deg; joints [33.744, -43.627, 116.123, 35.161, -74.66, -9.703]
  MoveC 1606 to (19.68, 383.04, -8.16) mm, rotated rx 180 ry 0 rz 0 deg; joints [33.728, -43.646, 116.147, 35.144, -74.66, -9.696] to (19.68, 382.85, -7.72) mm, rotated rx -180 ry 0 rz 0 deg; joints [33.721, -43.677, 116.161, 35.14, -74.645, -9.705]
  Set speed (1000.0 mm/s)
  MoveL 1607 to (19.68, 382.85, 6) mm, rotated rx 180 ry 0 rz 0 deg; joints [33.714, -44.524, 116.316, 35.244, -74.079, -10.117]
  MoveL 1608 to (-12.15, 384.12, 6) mm, rotated rx 180 ry 0 rz 0 deg; joints [33.023, -43.573, 113.992, 34.77, -72.825, -10.748]
  Set speed (25.4 mm/s)
  MoveL 1609 to (-12.15, 384.12, -4.36) mm, rotated rx 180 ry 0 rz 0 deg; joints [33.028, -42.95, 113.877, 34.687, -73.245, -10.446]
  MoveC 1610 to (-12.34, 384.12, -4.81) mm, rotated rx -180 ry 0 rz 0 deg; joints [33.024, -42.917, 113.858, 34.68, -73.255, -10.437] to (-12.79, 384.12, -5) mm, rotated rx -180 ry 0 rz 0 deg; joints [33.014, -42.893, 113.824, 34.672, -73.245, -10.44]
  Set speed (50.8 mm/s)
  MoveL 1611 to (-13.42, 384.12, -5) mm, rotated rx -180 ry 0 rz 0 deg; joints [33, -42.874, 113.778, 34.661, -73.22, -10.452]
  MoveC 1612 to (-13.87, 384.31, -5) mm, rotated rx 180 ry 0 rz 0 deg; joints [32.996, -42.858, 113.737, 34.662, -73.199, -10.465] to (-14.06, 384.76, -5) mm, rotated rx -180 ry 0 rz 0 deg; joints [33.007, -42.844, 113.703, 34.677, -73.184, -10.481]
  MoveL 1613 to (-14.06, 537.16, -5) mm, rotated rx -180 ry 0 rz 0 deg; joints [38.003, -39.719, 105.895, 40.74, -70.6, -15.014]
  MoveL 1614 to (-39.46, 537.16, -5) mm, rotated rx -180 ry 0 rz 0 deg; joints [37.401, -38.93, 104.049, 40.372, -69.636, -15.544]
  MoveC 1615 to (-52.16, 524.46, -5) mm, rotated rx 180 ry 0 rz 0 deg; joints [36.716, -38.819, 103.816, 39.698, -69.357, -15.392] to (-64.86, 537.16, -5) mm, rotated rx -180 ry 0 rz 0 deg; joints [36.815, -38.115, 102.159, 40.034, -68.652, -16.081]
  MoveL 1616 to (-90.26, 537.16, -5) mm, rotated rx 180 ry 0 rz 0 deg; joints [36.244, -37.275, 100.224, 39.726, -67.649, -16.628]
  MoveL 1617 to (-166.46, 537.16, -5) mm, rotated rx -180 ry 0 rz 0 deg; joints [34.621, -34.589, 94.12, 38.997, -64.511, -18.338]
  MoveC 1618 to (-179.16, 524.46, -5) mm, rotated rx -180 ry 0 rz 0 deg; joints [33.986, -34.429, 93.78, 38.383, -64.169, -18.183] to (-191.86, 537.16, -5) mm, rotated rx -180 ry 0 rz 0 deg; joints [34.109, -33.634, 91.977, 38.821, -63.42, -18.939]
  MoveL 1619 to (-293.46, 537.16, -5) mm, rotated rx 180 ry 0 rz 0 deg; joints [32.184, -29.458, 82.743, 38.506, -58.795, -21.582]
  MoveC 1620 to (-306.16, 524.46, -5) mm, rotated rx 180 ry 0 rz 0 deg; joints [31.595, -29.235, 82.273, 37.958, -58.382, -21.436] to (-318.86, 537.16, -5) mm, rotated rx -180 ry 0 rz 0 deg; joints [31.733, -28.311, 80.241, 38.539, -57.564, -22.324]
  MoveL 1621 to (-395.06, 537.16, -5) mm, rotated rx 180 ry 0 rz 0 deg; joints [30.446, -24.557, 72.129, 38.98, -53.644, -24.843]
  MoveL 1622 to (-420.46, 537.16, -5) mm, rotated rx -180 ry 0 rz 0 deg; joints [30.038, -23.179, 69.179, 39.267, -52.248, -25.814]
  MoveC 1623 to (-433.16, 524.46, -5) mm, rotated rx -180 ry 0 rz 0 deg; joints [29.488, -22.866, 68.524, 38.809, -51.742, -25.71] to (-445.86, 537.16, -5) mm, rotated rx -180 ry 0 rz 0 deg; joints [29.639, -21.724, 66.076, 39.644, -50.798, -26.875]
  MoveL 1624 to (-471.26, 537.16, -5) mm, rotated rx -180 ry 0 rz 0 deg; joints [29.25, -20.176, 62.792, 40.128, -49.284, -28.044]
  MoveL 1625 to (-471.26, 384.76, -5) mm, rotated rx -180 ry 0 rz 0 deg; joints [24.966, -24.674, 72.547, 32.509, -51.734, -20.861]
  MoveL 1626 to (-14.06, 384.76, -5) mm, rotated rx -180 ry 0 rz 0 deg; joints [33.007, -42.844, 113.703, 34.677, -73.184, -10.481]
  MoveC 1627 to (-13.61, 384.57, -5) mm, rotated rx 180 ry 0 rz 0 deg; joints [33.011, -42.861, 113.744, 34.677, -73.205, -10.467] to (-13.42, 384.12, -5) mm, rotated rx -180 ry 0 rz 0 deg; joints [33, -42.874, 113.778, 34.661, -73.22, -10.452]
  MoveL 1628 to (-13.42, 383.49, -5) mm, rotated rx 180 ry 0 rz 0 deg; joints [32.978, -42.886, 113.808, 34.636, -73.231, -10.435]
  MoveC 1629 to (-13.42, 383.04, -4.81) mm, rotated rx -180 ry 0 rz 0 deg; joints [32.962, -42.905, 113.831, 34.619, -73.231, -10.428] to (-13.42, 382.85, -4.37) mm, rotated rx -180 ry 0 rz 0 deg; joints [32.955, -42.935, 113.845, 34.615, -73.216, -10.436]
  Set speed (1000.0 mm/s)
  MoveL 1630 to (-13.42, 382.85, 5) mm, rotated rx -180 ry 0 rz 0 deg; joints [32.95, -43.499, 113.949, 34.69, -72.837, -10.708]
  MoveL 1631 to (-12.15, 384.12, 5) mm, rotated rx 180 ry 0 rz 0 deg; joints [33.023, -43.513, 113.981, 34.762, -72.866, -10.718]
  Set speed (25.4 mm/s)
  MoveL 1632 to (-12.15, 384.12, 1) mm, rotated rx -180 ry 0 rz 0 deg; joints [33.025, -43.273, 113.938, 34.729, -73.028, -10.601]
  MoveL 1633 to (-12.15, 384.12, -7.71) mm, rotated rx -180 ry 0 rz 0 deg; joints [33.03, -42.747, 113.838, 34.661, -73.379, -10.35]
  MoveC 1634 to (-12.34, 384.12, -8.16) mm, rotated rx -180 ry 0 rz 0 deg; joints [33.026, -42.715, 113.819, 34.654, -73.39, -10.34] to (-12.79, 384.12, -8.35) mm, rotated rx 180 ry 0 rz 0 deg; joints [33.016, -42.691, 113.785, 34.646, -73.379, -10.343]
  Set speed (50.8 mm/s)
  MoveL 1635 to (-13.42, 384.12, -8.35) mm, rotated rx 180 ry 0 rz 0 deg; joints [33.001, -42.672, 113.739, 34.635, -73.354, -10.356]
  MoveC 1636 to (-13.87, 384.31, -8.35) mm, rotated rx 180 ry 0 rz 0 deg; joints [32.998, -42.656, 113.698, 34.636, -73.333, -10.369] to (-14.06, 384.76, -8.35) mm, rotated rx 180 ry 0 rz 0 deg; joints [33.009, -42.642, 113.664, 34.651, -73.318, -10.385]
  MoveL 1637 to (-14.06, 537.16, -8.35) mm, rotated rx -180 ry 0 rz 0 deg; joints [38.005, -39.531, 105.856, 40.707, -70.714, -14.911]
  MoveL 1638 to (-39.46, 537.16, -8.35) mm, rotated rx -180 ry 0 rz 0 deg; joints [37.402, -38.745, 104.011, 40.338, -69.748, -15.444]
  MoveC 1639 to (-52.16, 524.46, -8.35) mm, rotated rx -180 ry 0 rz 0 deg; joints [36.718, -38.635, 103.778, 39.664, -69.47, -15.293] to (-64.86, 537.16, -8.35) mm, rotated rx 180 ry 0 rz 0 deg; joints [36.816, -37.934, 102.121, 39.999, -68.763, -15.983]
  MoveL 1640 to (-90.26, 537.16, -8.35) mm, rotated rx 180 ry 0 rz 0 deg; joints [36.246, -37.096, 100.186, 39.691, -67.758, -16.531]
  MoveL 1641 to (-166.46, 537.16, -8.35) mm, rotated rx -180 ry 0 rz 0 deg; joints [34.623, -34.418, 94.082, 38.958, -64.615, -18.245]
  MoveC 1642 to (-179.16, 524.46, -8.35) mm, rotated rx -180 ry 0 rz 0 deg; joints [33.988, -34.258, 93.742, 38.345, -64.274, -18.092] to (-191.86, 537.16, -8.35) mm, rotated rx -180 ry 0 rz 0 deg; joints [34.11, -33.465, 91.938, 38.782, -63.523, -18.848]
  MoveL 1643 to (-293.46, 537.16, -8.35) mm, rotated rx -180 ry 0 rz 0 deg; joints [32.186, -29.297, 82.703, 38.463, -58.89, -21.495]
  MoveC 1644 to (-306.16, 524.46, -8.35) mm, rotated rx 180 ry 0 rz 0 deg; joints [31.596, -29.075, 82.233, 37.914, -58.477, -21.35] to (-318.86, 537.16, -8.35) mm, rotated rx 180 ry 0 rz 0 deg; joints [31.735, -28.153, 80.2, 38.494, -57.657, -22.238]
  MoveL 1645 to (-395.06, 537.16, -8.35) mm, rotated rx 180 ry 0 rz 0 deg; joints [30.447, -24.403, 72.086, 38.93, -53.731, -24.758]
  MoveL 1646 to (-420.46, 537.16, -8.35) mm, rotated rx -180 ry 0 rz 0 deg; joints [30.039, -23.027, 69.135, 39.216, -52.332, -25.729]
  MoveC 1647 to (-433.16, 524.46, -8.35) mm, rotated rx 180 ry 0 rz 0 deg; joints [29.49, -22.714, 68.48, 38.758, -51.826, -25.625] to (-445.86, 537.16, -8.35) mm, rotated rx -180 ry 0 rz 0 deg; joints [29.64, -21.572, 66.03, 39.591, -50.879, -26.789]
  MoveL 1648 to (-471.26, 537.16, -8.35) mm, rotated rx -180 ry 0 rz 0 deg; joints [29.251, -20.026, 62.744, 40.073, -49.363, -27.958]
  MoveL 1649 to (-471.26, 384.76, -8.35) mm, rotated rx -180 ry 0 rz 0 deg; joints [24.967, -24.52, 72.504, 32.464, -51.828, -20.786]
  MoveL 1650 to (-14.06, 384.76, -8.35) mm, rotated rx -180 ry 0 rz 0 deg; joints [33.009, -42.642, 113.664, 34.651, -73.318, -10.385]
  MoveC 1651 to (-13.61, 384.57, -8.35) mm, rotated rx -180 ry 0 rz 0 deg; joints [33.013, -42.659, 113.705, 34.651, -73.339, -10.371] to (-13.42, 384.12, -8.35) mm, rotated rx 180 ry 0 rz 0 deg; joints [33.001, -42.672, 113.739, 34.635, -73.354, -10.356]
  MoveL 1652 to (-13.42, 383.49, -8.35) mm, rotated rx -180 ry 0 rz 0 deg; joints [32.979, -42.684, 113.769, 34.61, -73.365, -10.339]
  MoveC 1653 to (-13.42, 383.04, -8.16) mm, rotated rx -180 ry 0 rz 0 deg; joints [32.963, -42.703, 113.792, 34.593, -73.365, -10.332] to (-13.42, 382.85, -7.72) mm, rotated rx 180 ry 0 rz 0 deg; joints [32.957, -42.733, 113.806, 34.589, -73.351, -10.34]
  Set speed (1000.0 mm/s)
  MoveL 1654 to (-13.42, 382.85, 15) mm, rotated rx -180 ry 0 rz 0 deg; joints [32.945, -44.098, 114.052, 34.773, -72.429, -11.002]
  MoveL 1655 to (-13.42, 382.85, 15) mm, rotated rx -180 ry 0 rz 0 deg; joints [32.945, -44.098, 114.052, 34.773, -72.429, -11.002]
